LIN {X 0,Y 687.09,Z 992.261,A -85,B 0,C 180,E1 4203.082,E2 4203.082} C_VEL
LIN {X 0,Y 685.189,Z 1030.592,A -85,B 0,C 180,E1 4205.694,E2 4205.694} C_VEL
LIN {X 0,Y 683.437,Z 1066.226,A -85,B 0,C 180,E1 4208.838,E2 4208.838} C_VEL
LIN {X 0,Y 682.212,Z 1095.925,A -85,B 0,C 180,E1 4212.224,E2 4212.224} C_VEL
LIN {X 0,Y 681.417,Z 1120.366,A -85,B 0,C 180,E1 4215.88,E2 4215.88} C_VEL
LIN {X 0,Y 680.982,Z 1137.956,A -85,B 0,C 180,E1 4219.451,E2 4219.451} C_VEL
LIN {X 0,Y 680.83,Z 1150.116,A -85,B 0,C 180,E1 4222.988,E2 4222.988} C_VEL
LIN {X 0,Y 680.781,Z 1156.664,A -85,B 0,C 180,E1 4226.181,E2 4226.181} C_VEL
LIN {X 0,Y 680.724,Z 1159.5,A -85,B 0,C 180,E1 4229.999,E2 4229.999} C_VEL
LIN {X 0,Y 680.746,Z 1156.667,A -85,B 0,C 180,E1 4233.818,E2 4233.818} C_VEL
LIN {X 0,Y 680.9,Z 1150.12,A -85,B 0,C 180,E1 4237.01,E2 4237.01} C_VEL
LIN {X 0,Y 681.026,Z 1137.964,A -85,B 0,C 180,E1 4240.547,E2 4240.547} C_VEL
LIN {X 0,Y 681.455,Z 1120.372,A -85,B 0,C 180,E1 4244.117,E2 4244.117} C_VEL
LIN {X 0,Y 682.306,Z 1095.708,A -85,B 0,C 180,E1 4247.801,E2 4247.801} C_VEL
LIN {X 0,Y 683.582,Z 1064.828,A -85,B 0,C 180,E1 4251.298,E2 4251.298} C_VEL
LIN {X 0,Y 685.214,Z 1030.571,A -85,B 0,C 180,E1 4254.307,E2 4254.307} C_VEL
LIN {X 0,Y 687.123,Z 990.6,A -85,B 0,C 180,E1 4257.023,E2 4257.023} C_VEL
LIN {X 0,Y 689.048,Z 948.933,A -85,B 0,C 180,E1 4259.157,E2 4259.157} C_VEL
LIN {X 0,Y 690.718,Z 906.278,A -85,B 0,C 180,E1 4260.75,E2 4260.75} C_VEL
LIN {X 0,Y 691.991,Z 863.04,A -85,B 0,C 180,E1 4261.837,E2 4261.837} C_VEL
LIN {X 0,Y 691.945,Z 806.371,A -85,B 0,C 180,E1 4262.655,E2 4262.655} C_VEL
LIN {X 0,Y 680.359,Z 780.81,A -85,B 0,C 180,E1 4263.619,E2 4263.619} C_VEL
LIN {X 0,Y 680.153,Z 780.81,A -85,B 0,C 180,E1 4268.974,E2 4268.974} C_VEL
LIN {X 0,Y 680.422,Z 780.81,A -85,B 0,C 180,E1 4273.507,E2 4273.507} C_VEL
LIN {X 0,Y 680.172,Z 780.81,A -85,B 0,C 180,E1 4279.056,E2 4279.056} C_VEL
LIN {X 0,Y 680.227,Z 780.81,A -85,B 0,C 180,E1 4283.154,E2 4283.154} C_VEL
LIN {X 0,Y 680.191,Z 780.81,A -85,B 0,C 180,E1 4287.788,E2 4287.788} C_VEL
LIN {X 0,Y 680.45,Z 780.81,A -85,B 0,C 180,E1 4292.658,E2 4292.658} C_VEL
LIN {X 0,Y 680.425,Z 780.81,A -85,B 0,C 180,E1 4297.825,E2 4297.825} C_VEL
LIN {X 0,Y 680.516,Z 780.81,A -85,B 0,C 180,E1 4303.227,E2 4303.227} C_VEL
LIN {X 0,Y 680.543,Z 780.81,A -85,B 0,C 180,E1 4308.476,E2 4308.476} C_VEL
LIN {X 0,Y 680.684,Z 780.81,A -85,B 0,C 180,E1 4313.63,E2 4313.63} C_VEL
LIN {X 0,Y 680.631,Z 780.81,A -85,B 0,C 180,E1 4318.73,E2 4318.73} C_VEL
LIN {X 0,Y 680.66,Z 780.81,A -85,B 0,C 180,E1 4322.546,E2 4322.546} C_VEL
LIN {X 0,Y 680.609,Z 780.81,A -85,B 0,C 180,E1 4326.374,E2 4326.374} C_VEL
LIN {X 0,Y 680.539,Z 780.81,A -85,B 0,C 180,E1 4331.528,E2 4331.528} C_VEL
LIN {X 0,Y 680.552,Z 780.81,A -85,B 0,C 180,E1 4336.776,E2 4336.776} C_VEL
LIN {X 0,Y 680.385,Z 780.81,A -85,B 0,C 180,E1 4342.181,E2 4342.181} C_VEL
LIN {X 0,Y 680.369,Z 780.81,A -85,B 0,C 180,E1 4347.328,E2 4347.328} C_VEL
LIN {X 0,Y 680.311,Z 780.81,A -85,B 0,C 180,E1 4352.431,E2 4352.431} C_VEL
LIN {X 0,Y 680.211,Z 780.81,A -85,B 0,C 180,E1 4356.895,E2 4356.895} C_VEL
LIN {X 0,Y 680.321,Z 780.81,A -85,B 0,C 180,E1 4362.864,E2 4362.864} C_VEL
LIN {X 0,Y 680.144,Z 780.81,A -85,B 0,C 180,E1 4368.202,E2 4368.202} C_VEL
LIN {X 0,Y 680.322,Z 780.81,A -85,B 0,C 180,E1 4373.152,E2 4373.152} C_VEL
LIN {X 0,Y 680.408,Z 781.584,A -85,B 0,C 180,E1 4373.863,E2 4373.863} C_VEL
LIN {X 0,Y 692.3,Z 808.432,A -85,B 0,C 180,E1 4374.861,E2 4374.861} C_VEL
LIN {X 0,Y 691.206,Z 854.71,A -85,B 0,C 180,E1 4375.867,E2 4375.867} C_VEL
LIN {X 0,Y 689.535,Z 897.482,A -85,B 0,C 180,E1 4377.317,E2 4377.317} C_VEL
LIN {X 0,Y 687.817,Z 937.086,A -85,B 0,C 180,E1 4379.173,E2 4379.173} C_VEL
LIN {X 0,Y 685.919,Z 976.276,A -85,B 0,C 180,E1 4381.593,E2 4381.593} C_VEL
LIN {X 0,Y 684.097,Z 1013.54,A -85,B 0,C 180,E1 4384.581,E2 4384.581} C_VEL
LIN {X 0,Y 682.642,Z 1045.528,A -85,B 0,C 180,E1 4387.895,E2 4387.895} C_VEL
LIN {X 0,Y 681.64,Z 1071.691,A -85,B 0,C 180,E1 4391.418,E2 4391.418} C_VEL
LIN {X 0,Y 681.199,Z 1089.618,A -85,B 0,C 180,E1 4394.563,E2 4394.563} C_VEL
LIN {X 0,Y 680.932,Z 1103.952,A -85,B 0,C 180,E1 4397.975,E2 4397.975} C_VEL
LIN {X 0,Y 680.821,Z 1112.845,A -85,B 0,C 180,E1 4401.063,E2 4401.063} C_VEL
LIN {X 0,Y 680.722,Z 1118.621,A -85,B 0,C 180,E1 4404.906,E2 4404.906} C_VEL
LIN {X 0,Y 680.773,Z 1119.375,A -85,B 0,C 180,E1 4407.456,E2 4407.456} C_VEL
LIN {X 0,Y 680.825,Z 1115.946,A -85,B 0,C 180,E1 4411.273,E2 4411.273} C_VEL
LIN {X 0,Y 680.875,Z 1106.765,A -85,B 0,C 180,E1 4415.094,E2 4415.094} C_VEL
LIN {X 0,Y 681.054,Z 1093.102,A -85,B 0,C 180,E1 4418.614,E2 4418.614} C_VEL
LIN {X 0,Y 681.647,Z 1073.872,A -85,B 0,C 180,E1 4422.158,E2 4422.158} C_VEL
LIN {X 0,Y 682.563,Z 1047.417,A -85,B 0,C 180,E1 4425.79,E2 4425.79} C_VEL
LIN {X 0,Y 683.892,Z 1016.827,A -85,B 0,C 180,E1 4429.021,E2 4429.021} C_VEL
LIN {X 0,Y 685.562,Z 982.863,A -85,B 0,C 180,E1 4431.837,E2 4431.837} C_VEL
LIN {X 0,Y 687.416,Z 945.41,A -85,B 0,C 180,E1 4434.273,E2 4434.273} C_VEL
LIN {X 0,Y 689.372,Z 903.344,A -85,B 0,C 180,E1 4436.353,E2 4436.353} C_VEL
LIN {X 0,Y 691.019,Z 860.946,A -85,B 0,C 180,E1 4437.864,E2 4437.864} C_VEL
LIN {X 0,Y 692.216,Z 820.938,A -85,B 0,C 180,E1 4438.82,E2 4438.82} C_VEL
LIN {X 0,Y 691.723,Z 806.397,A -85,B 0,C 180,E1 4439.108,E2 4439.108} C_VEL
LIN {X 0,Y 680.353,Z 780.81,A -85,B 0,C 180,E1 4440.141,E2 4440.141} C_VEL
LIN {X 0,Y 680.26,Z 780.81,A -85,B 0,C 180,E1 4445.28,E2 4445.28} C_VEL
LIN {X 0,Y 680.117,Z 780.81,A -85,B 0,C 180,E1 4450.946,E2 4450.946} C_VEL
LIN {X 0,Y 680.316,Z 780.81,A -85,B 0,C 180,E1 4455.299,E2 4455.299} C_VEL
LIN {X 0,Y 680.19,Z 780.81,A -85,B 0,C 180,E1 4461.039,E2 4461.039} C_VEL
LIN {X 0,Y 680.175,Z 780.81,A -85,B 0,C 180,E1 4466.265,E2 4466.265} C_VEL
LIN {X 0,Y 680.318,Z 780.81,A -85,B 0,C 180,E1 4470.751,E2 4470.751} C_VEL
LIN {X 0,Y 680.406,Z 780.81,A -85,B 0,C 180,E1 4475.585,E2 4475.585} C_VEL
LIN {X 0,Y 680.489,Z 780.81,A -85,B 0,C 180,E1 4480.545,E2 4480.545} C_VEL
LIN {X 0,Y 680.5,Z 780.81,A -85,B 0,C 180,E1 4485.862,E2 4485.862} C_VEL
LIN {X 0,Y 680.619,Z 780.81,A -85,B 0,C 180,E1 4491.059,E2 4491.059} C_VEL
LIN {X 0,Y 680.741,Z 780.81,A -85,B 0,C 180,E1 4496.18,E2 4496.18} C_VEL
LIN {X 0,Y 680.88,Z 780.81,A -85,B 0,C 180,E1 4501.27,E2 4501.27} C_VEL
LIN {X 0,Y 680.579,Z 780.81,A -85,B 0,C 180,E1 4506.371,E2 4506.371} C_VEL
LIN {X 0,Y 680.539,Z 780.81,A -85,B 0,C 180,E1 4511.524,E2 4511.524} C_VEL
LIN {X 0,Y 680.564,Z 780.81,A -85,B 0,C 180,E1 4516.772,E2 4516.772} C_VEL
LIN {X 0,Y 680.422,Z 780.81,A -85,B 0,C 180,E1 4522.175,E2 4522.175} C_VEL
LIN {X 0,Y 680.366,Z 780.81,A -85,B 0,C 180,E1 4522.914,E2 4522.914} C_VEL
LIN {X 0,Y 676.415,Z 780.81,A -85,B 0,C 180,E1 4524.348,E2 4524.348} C_VEL
LIN {X 0,Y 672.467,Z 780.81,A -85,B 0,C 180,E1 4525.798,E2 4525.798} C_VEL
LIN {X 0,Y 672.401,Z 780.81,A -85,B 0,C 180,E1 4531.351,E2 4531.351} C_VEL
LIN {X 0,Y 672.326,Z 780.81,A -85,B 0,C 180,E1 4535.988,E2 4535.988} C_VEL
LIN {X 0,Y 672.186,Z 780.81,A -85,B 0,C 180,E1 4540.676,E2 4540.676} C_VEL
LIN {X 0,Y 672.254,Z 780.81,A -85,B 0,C 180,E1 4545.984,E2 4545.984} C_VEL
LIN {X 0,Y 672.227,Z 780.81,A -85,B 0,C 180,E1 4550.992,E2 4550.992} C_VEL
LIN {X 0,Y 672.468,Z 781.462,A -85,B 0,C 180,E1 4555.963,E2 4555.963} C_VEL
LIN {X 0,Y 685.899,Z 811.043,A -85,B 0,C 180,E1 4557.078,E2 4557.078} C_VEL
LIN {X 0,Y 685.2,Z 867.047,A -85,B 0,C 180,E1 4557.895,E2 4557.895} C_VEL
LIN {X 0,Y 683.792,Z 911.293,A -85,B 0,C 180,E1 4559.07,E2 4559.07} C_VEL
LIN {X 0,Y 681.813,Z 953.795,A -85,B 0,C 180,E1 4560.736,E2 4560.736} C_VEL
LIN {X 0,Y 679.857,Z 992.661,A -85,B 0,C 180,E1 4562.798,E2 4562.798} C_VEL
LIN {X 0,Y 677.754,Z 1031.108,A -85,B 0,C 180,E1 4565.453,E2 4565.453} C_VEL
LIN {X 0,Y 675.905,Z 1065.391,A -85,B 0,C 180,E1 4568.503,E2 4568.503} C_VEL
LIN {X 0,Y 674.501,Z 1095.923,A -85,B 0,C 180,E1 4572.014,E2 4572.014} C_VEL
LIN {X 0,Y 673.612,Z 1120.364,A -85,B 0,C 180,E1 4575.713,E2 4575.713} C_VEL
LIN {X 0,Y 673.147,Z 1136.615,A -85,B 0,C 180,E1 4578.999,E2 4578.999} C_VEL
LIN {X 0,Y 672.935,Z 1148.221,A -85,B 0,C 180,E1 4582.256,E2 4582.256} C_VEL
LIN {X 0,Y 672.913,Z 1155.686,A -85,B 0,C 180,E1 4585.491,E2 4585.491} C_VEL
LIN {X 0,Y 672.874,Z 1159.169,A -85,B 0,C 180,E1 4588.712,E2 4588.712} C_VEL
LIN {X 0,Y 672.847,Z 1158.224,A -85,B 0,C 180,E1 4592.574,E2 4592.574} C_VEL
LIN {X 0,Y 672.976,Z 1153.237,A -85,B 0,C 180,E1 4595.799,E2 4595.799} C_VEL
LIN {X 0,Y 673.038,Z 1141.814,A -85,B 0,C 180,E1 4599.693,E2 4599.693} C_VEL
LIN {X 0,Y 673.402,Z 1127.472,A -85,B 0,C 180,E1 4602.967,E2 4602.967} C_VEL
LIN {X 0,Y 674.051,Z 1105.875,A -85,B 0,C 180,E1 4606.608,E2 4606.608} C_VEL
LIN {X 0,Y 675.147,Z 1079.569,A -85,B 0,C 180,E1 4609.975,E2 4609.975} C_VEL
LIN {X 0,Y 676.765,Z 1049.45,A -85,B 0,C 180,E1 4613,E2 4613} C_VEL
LIN {X 0,Y 678.651,Z 1014.986,A -85,B 0,C 180,E1 4615.744,E2 4615.744} C_VEL
LIN {X 0,Y 680.85,Z 974.62,A -85,B 0,C 180,E1 4618.232,E2 4618.232} C_VEL
LIN {X 0,Y 682.963,Z 931.607,A -85,B 0,C 180,E1 4620.204,E2 4620.204} C_VEL
LIN {X 0,Y 684.568,Z 890.233,A -85,B 0,C 180,E1 4621.55,E2 4621.55} C_VEL
LIN {X 0,Y 685.646,Z 849.593,A -85,B 0,C 180,E1 4622.422,E2 4622.422} C_VEL
LIN {X 0,Y 685.428,Z 809.206,A -85,B 0,C 180,E1 4622.97,E2 4622.97} C_VEL
LIN {X 0,Y 672.415,Z 780.81,A -85,B 0,C 180,E1 4624.066,E2 4624.066} C_VEL
LIN {X 0,Y 672.257,Z 780.81,A -85,B 0,C 180,E1 4629.004,E2 4629.004} C_VEL
LIN {X 0,Y 672.483,Z 780.81,A -85,B 0,C 180,E1 4634.153,E2 4634.153} C_VEL
LIN {X 0,Y 672.314,Z 780.81,A -85,B 0,C 180,E1 4639.834,E2 4639.834} C_VEL
LIN {X 0,Y 672.292,Z 780.81,A -85,B 0,C 180,E1 4644.249,E2 4644.249} C_VEL
LIN {X 0,Y 672.295,Z 780.81,A -85,B 0,C 180,E1 4648.879,E2 4648.879} C_VEL
LIN {X 0,Y 672.521,Z 780.81,A -85,B 0,C 180,E1 4653.995,E2 4653.995} C_VEL
LIN {X 0,Y 672.529,Z 780.81,A -85,B 0,C 180,E1 4658.936,E2 4658.936} C_VEL
LIN {X 0,Y 672.629,Z 780.81,A -85,B 0,C 180,E1 4664.365,E2 4664.365} C_VEL
LIN {X 0,Y 672.708,Z 780.81,A -85,B 0,C 180,E1 4669.651,E2 4669.651} C_VEL
LIN {X 0,Y 672.703,Z 780.81,A -85,B 0,C 180,E1 4674.848,E2 4674.848} C_VEL
LIN {X 0,Y 672.744,Z 780.81,A -85,B 0,C 180,E1 4678.715,E2 4678.715} C_VEL
LIN {X 0,Y 672.758,Z 780.81,A -85,B 0,C 180,E1 4682.576,E2 4682.576} C_VEL
LIN {X 0,Y 672.702,Z 780.81,A -85,B 0,C 180,E1 4686.45,E2 4686.45} C_VEL
LIN {X 0,Y 672.681,Z 780.81,A -85,B 0,C 180,E1 4690.353,E2 4690.353} C_VEL
LIN {X 0,Y 672.653,Z 780.81,A -85,B 0,C 180,E1 4695.638,E2 4695.638} C_VEL
LIN {X 0,Y 672.522,Z 780.81,A -85,B 0,C 180,E1 4701.068,E2 4701.068} C_VEL
LIN {X 0,Y 672.434,Z 780.81,A -85,B 0,C 180,E1 4706.705,E2 4706.705} C_VEL
LIN {X 0,Y 672.359,Z 780.81,A -85,B 0,C 180,E1 4711.348,E2 4711.348} C_VEL
LIN {X 0,Y 672.303,Z 780.81,A -85,B 0,C 180,E1 4715.988,E2 4715.988} C_VEL
LIN {X 0,Y 672.208,Z 780.81,A -85,B 0,C 180,E1 4720.68,E2 4720.68} C_VEL
LIN {X 0,Y 672.349,Z 780.81,A -85,B 0,C 180,E1 4725.981,E2 4725.981} C_VEL
LIN {X 0,Y 672.42,Z 780.81,A -85,B 0,C 180,E1 4731.854,E2 4731.854} C_VEL
LIN {X 0,Y 672.432,Z 780.81,A -85,B 0,C 180,E1 4733.398,E2 4733.398} C_VEL
LIN {X 0,Y 685.61,Z 812.911,A -85,B 0,C 180,E1 4734.594,E2 4734.594} C_VEL
LIN {X 0,Y 684.35,Z 856.364,A -85,B 0,C 180,E1 4735.567,E2 4735.567} C_VEL
LIN {X 0,Y 682.476,Z 899.679,A -85,B 0,C 180,E1 4737.073,E2 4737.073} C_VEL
LIN {X 0,Y 680.432,Z 940.833,A -85,B 0,C 180,E1 4739.065,E2 4739.065} C_VEL
LIN {X 0,Y 678.453,Z 978.628,A -85,B 0,C 180,E1 4741.469,E2 4741.469} C_VEL
LIN {X 0,Y 676.521,Z 1014.57,A -85,B 0,C 180,E1 4744.413,E2 4744.413} C_VEL
LIN {X 0,Y 674.916,Z 1046.522,A -85,B 0,C 180,E1 4747.785,E2 4747.785} C_VEL
LIN {X 0,Y 673.823,Z 1072.54,A -85,B 0,C 180,E1 4751.364,E2 4751.364} C_VEL
LIN {X 0,Y 673.302,Z 1091.329,A -85,B 0,C 180,E1 4754.78,E2 4754.78} C_VEL
LIN {X 0,Y 673.042,Z 1105.621,A -85,B 0,C 180,E1 4758.343,E2 4758.343} C_VEL
LIN {X 0,Y 672.916,Z 1115.336,A -85,B 0,C 180,E1 4762.257,E2 4762.257} C_VEL
LIN {X 0,Y 672.898,Z 1119.294,A -85,B 0,C 180,E1 4766.138,E2 4766.138} C_VEL
LIN {X 0,Y 672.908,Z 1117.744,A -85,B 0,C 180,E1 4770.001,E2 4770.001} C_VEL
LIN {X 0,Y 673.061,Z 1110.564,A -85,B 0,C 180,E1 4773.863,E2 4773.863} C_VEL
LIN {X 0,Y 673.213,Z 1097.492,A -85,B 0,C 180,E1 4777.741,E2 4777.741} C_VEL
LIN {X 0,Y 673.691,Z 1079.897,A -85,B 0,C 180,E1 4781.319,E2 4781.319} C_VEL
LIN {X 0,Y 674.447,Z 1056.011,A -85,B 0,C 180,E1 4784.932,E2 4784.932} C_VEL
LIN {X 0,Y 675.9,Z 1025.8,A -85,B 0,C 180,E1 4788.409,E2 4788.409} C_VEL
LIN {X 0,Y 677.806,Z 990.093,A -85,B 0,C 180,E1 4791.584,E2 4791.584} C_VEL
LIN {X 0,Y 679.981,Z 950.7,A -85,B 0,C 180,E1 4794.278,E2 4794.278} C_VEL
LIN {X 0,Y 682.058,Z 909.948,A -85,B 0,C 180,E1 4796.391,E2 4796.391} C_VEL
LIN {X 0,Y 683.81,Z 870.24,A -85,B 0,C 180,E1 4797.919,E2 4797.919} C_VEL
LIN {X 0,Y 685.308,Z 826.609,A -85,B 0,C 180,E1 4799.065,E2 4799.065} C_VEL
LIN {X 0,Y 684.896,Z 808.687,A -85,B 0,C 180,E1 4799.434,E2 4799.434} C_VEL
LIN {X 0,Y 672.411,Z 780.81,A -85,B 0,C 180,E1 4800.538,E2 4800.538} C_VEL
LIN {X 0,Y 672.289,Z 780.81,A -85,B 0,C 180,E1 4805.762,E2 4805.762} C_VEL
LIN {X 0,Y 672.207,Z 780.81,A -85,B 0,C 180,E1 4810.687,E2 4810.687} C_VEL
LIN {X 0,Y 672.336,Z 780.81,A -85,B 0,C 180,E1 4815.841,E2 4815.841} C_VEL
LIN {X 0,Y 672.293,Z 780.81,A -85,B 0,C 180,E1 4821.003,E2 4821.003} C_VEL
LIN {X 0,Y 672.283,Z 780.81,A -85,B 0,C 180,E1 4826.271,E2 4826.271} C_VEL
LIN {X 0,Y 672.462,Z 780.81,A -85,B 0,C 180,E1 4831.846,E2 4831.846} C_VEL
LIN {X 0,Y 672.461,Z 780.81,A -85,B 0,C 180,E1 4837.122,E2 4837.122} C_VEL
LIN {X 0,Y 672.59,Z 780.81,A -85,B 0,C 180,E1 4841.668,E2 4841.668} C_VEL
LIN {X 0,Y 672.588,Z 780.81,A -85,B 0,C 180,E1 4845.692,E2 4845.692} C_VEL
LIN {X 0,Y 672.713,Z 780.81,A -85,B 0,C 180,E1 4851.256,E2 4851.256} C_VEL
LIN {X 0,Y 672.831,Z 780.81,A -85,B 0,C 180,E1 4856.135,E2 4856.135} C_VEL
LIN {X 0,Y 672.979,Z 780.81,A -85,B 0,C 180,E1 4861.284,E2 4861.284} C_VEL
LIN {X 0,Y 672.674,Z 780.81,A -85,B 0,C 180,E1 4866.446,E2 4866.446} C_VEL
LIN {X 0,Y 672.669,Z 780.81,A -85,B 0,C 180,E1 4870.349,E2 4870.349} C_VEL
LIN {X 0,Y 672.647,Z 780.81,A -85,B 0,C 180,E1 4875.635,E2 4875.635} C_VEL
LIN {X 0,Y 672.572,Z 780.81,A -85,B 0,C 180,E1 4881.062,E2 4881.062} C_VEL
LIN {X 0,Y 672.467,Z 780.81,A -85,B 0,C 180,E1 4885.798,E2 4885.798} C_VEL
LIN {X 0,Y 668.561,Z 780.81,A -85,B 0,C 180,E1 4887.256,E2 4887.256} C_VEL
LIN {X 0,Y 664.506,Z 780.81,A -85,B 0,C 180,E1 4888.73,E2 4888.73} C_VEL
LIN {X 0,Y 664.534,Z 780.81,A -85,B 0,C 180,E1 4893.067,E2 4893.067} C_VEL
LIN {X 0,Y 664.329,Z 780.81,A -85,B 0,C 180,E1 4897.88,E2 4897.88} C_VEL
LIN {X 0,Y 664.274,Z 780.81,A -85,B 0,C 180,E1 4903.285,E2 4903.285} C_VEL
LIN {X 0,Y 664.27,Z 780.81,A -85,B 0,C 180,E1 4908.722,E2 4908.722} C_VEL
LIN {X 0,Y 664.417,Z 780.81,A -85,B 0,C 180,E1 4913.748,E2 4913.748} C_VEL
LIN {X 0,Y 664.48,Z 780.81,A -85,B 0,C 180,E1 4915.49,E2 4915.49} C_VEL
LIN {X 0,Y 679.318,Z 813.462,A -85,B 0,C 180,E1 4916.747,E2 4916.747} C_VEL
LIN {X 0,Y 678.502,Z 867.045,A -85,B 0,C 180,E1 4917.539,E2 4917.539} C_VEL
LIN {X 0,Y 676.925,Z 911.802,A -85,B 0,C 180,E1 4918.739,E2 4918.739} C_VEL
LIN {X 0,Y 674.776,Z 954.064,A -85,B 0,C 180,E1 4920.414,E2 4920.414} C_VEL
LIN {X 0,Y 672.573,Z 994.032,A -85,B 0,C 180,E1 4922.568,E2 4922.568} C_VEL
LIN {X 0,Y 670.323,Z 1031.236,A -85,B 0,C 180,E1 4925.173,E2 4925.173} C_VEL
LIN {X 0,Y 668.273,Z 1066.264,A -85,B 0,C 180,E1 4928.338,E2 4928.338} C_VEL
LIN {X 0,Y 666.779,Z 1096.55,A -85,B 0,C 180,E1 4931.882,E2 4931.882} C_VEL
LIN {X 0,Y 665.808,Z 1120.363,A -85,B 0,C 180,E1 4935.542,E2 4935.542} C_VEL
LIN {X 0,Y 665.248,Z 1137.958,A -85,B 0,C 180,E1 4939.198,E2 4939.198} C_VEL
LIN {X 0,Y 665.055,Z 1150.116,A -85,B 0,C 180,E1 4942.82,E2 4942.82} C_VEL
LIN {X 0,Y 664.989,Z 1156.663,A -85,B 0,C 180,E1 4946.09,E2 4946.09} C_VEL
LIN {X 0,Y 664.947,Z 1159.5,A -85,B 0,C 180,E1 4949.999,E2 4949.999} C_VEL
LIN {X 0,Y 664.964,Z 1156.666,A -85,B 0,C 180,E1 4953.908,E2 4953.908} C_VEL
LIN {X 0,Y 665.132,Z 1150.12,A -85,B 0,C 180,E1 4957.177,E2 4957.177} C_VEL
LIN {X 0,Y 665.406,Z 1136.623,A -85,B 0,C 180,E1 4961.129,E2 4961.129} C_VEL
LIN {X 0,Y 665.961,Z 1118.841,A -85,B 0,C 180,E1 4964.717,E2 4964.717} C_VEL
LIN {X 0,Y 666.903,Z 1095.045,A -85,B 0,C 180,E1 4968.311,E2 4968.311} C_VEL
LIN {X 0,Y 668.399,Z 1064.744,A -85,B 0,C 180,E1 4971.815,E2 4971.815} C_VEL
LIN {X 0,Y 670.485,Z 1029.076,A -85,B 0,C 180,E1 4974.997,E2 4974.997} C_VEL
LIN {X 0,Y 672.77,Z 990.127,A -85,B 0,C 180,E1 4977.678,E2 4977.678} C_VEL
LIN {X 0,Y 675.203,Z 947.105,A -85,B 0,C 180,E1 4979.903,E2 4979.903} C_VEL
LIN {X 0,Y 677.144,Z 904.152,A -85,B 0,C 180,E1 4981.507,E2 4981.507} C_VEL
LIN {X 0,Y 678.642,Z 860.929,A -85,B 0,C 180,E1 4982.58,E2 4982.58} C_VEL
LIN {X 0,Y 678.651,Z 811.393,A -85,B 0,C 180,E1 4983.315,E2 4983.315} C_VEL
LIN {X 0,Y 664.443,Z 780.81,A -85,B 0,C 180,E1 4984.511,E2 4984.511} C_VEL
LIN {X 0,Y 664.333,Z 780.81,A -85,B 0,C 180,E1 4989.56,E2 4989.56} C_VEL
LIN {X 0,Y 664.474,Z 780.81,A -85,B 0,C 180,E1 4994.827,E2 4994.827} C_VEL
LIN {X 0,Y 664.395,Z 780.81,A -85,B 0,C 180,E1 5000.65,E2 5000.65} C_VEL
LIN {X 0,Y 664.346,Z 780.81,A -85,B 0,C 180,E1 5005.354,E2 5005.354} C_VEL
LIN {X 0,Y 664.408,Z 780.81,A -85,B 0,C 180,E1 5009.984,E2 5009.984} C_VEL
LIN {X 0,Y 664.606,Z 780.81,A -85,B 0,C 180,E1 5014.412,E2 5014.412} C_VEL
LIN {X 0,Y 664.627,Z 780.81,A -85,B 0,C 180,E1 5020.065,E2 5020.065} C_VEL
LIN {X 0,Y 664.658,Z 780.81,A -85,B 0,C 180,E1 5025.522,E2 5025.522} C_VEL
LIN {X 0,Y 664.759,Z 780.81,A -85,B 0,C 180,E1 5030.848,E2 5030.848} C_VEL
LIN {X 0,Y 664.919,Z 780.81,A -85,B 0,C 180,E1 5036.093,E2 5036.093} C_VEL
LIN {X 0,Y 665.057,Z 780.81,A -85,B 0,C 180,E1 5041.333,E2 5041.333} C_VEL
LIN {X 0,Y 664.802,Z 780.81,A -85,B 0,C 180,E1 5046.527,E2 5046.527} C_VEL
LIN {X 0,Y 664.723,Z 780.81,A -85,B 0,C 180,E1 5051.806,E2 5051.806} C_VEL
LIN {X 0,Y 664.702,Z 780.81,A -85,B 0,C 180,E1 5057.293,E2 5057.293} C_VEL
LIN {X 0,Y 664.539,Z 780.81,A -85,B 0,C 180,E1 5062.739,E2 5062.739} C_VEL
LIN {X 0,Y 664.503,Z 780.81,A -85,B 0,C 180,E1 5067.519,E2 5067.519} C_VEL
LIN {X 0,Y 664.506,Z 780.81,A -85,B 0,C 180,E1 5073.073,E2 5073.073} C_VEL
LIN {X 0,Y 664.317,Z 780.81,A -85,B 0,C 180,E1 5077.886,E2 5077.886} C_VEL
LIN {X 0,Y 664.433,Z 780.81,A -85,B 0,C 180,E1 5083.301,E2 5083.301} C_VEL
LIN {X 0,Y 664.315,Z 780.81,A -85,B 0,C 180,E1 5088.727,E2 5088.727} C_VEL
LIN {X 0,Y 664.51,Z 780.81,A -85,B 0,C 180,E1 5092.933,E2 5092.933} C_VEL
LIN {X 0,Y 678.862,Z 813.526,A -85,B 0,C 180,E1 5094.244,E2 5094.244} C_VEL
LIN {X 0,Y 677.544,Z 857.036,A -85,B 0,C 180,E1 5095.234,E2 5095.234} C_VEL
LIN {X 0,Y 675.456,Z 901.471,A -85,B 0,C 180,E1 5096.808,E2 5096.808} C_VEL
LIN {X 0,Y 673.206,Z 942.54,A -85,B 0,C 180,E1 5098.841,E2 5098.841} C_VEL
LIN {X 0,Y 671.047,Z 979.928,A -85,B 0,C 180,E1 5101.269,E2 5101.269} C_VEL
LIN {X 0,Y 668.947,Z 1015.39,A -85,B 0,C 180,E1 5104.225,E2 5104.225} C_VEL
LIN {X 0,Y 667.242,Z 1046.933,A -85,B 0,C 180,E1 5107.608,E2 5107.608} C_VEL
LIN {X 0,Y 666.017,Z 1073.389,A -85,B 0,C 180,E1 5111.309,E2 5111.309} C_VEL
LIN {X 0,Y 665.453,Z 1091.617,A -85,B 0,C 180,E1 5114.696,E2 5114.696} C_VEL
LIN {X 0,Y 665.154,Z 1105.491,A -85,B 0,C 180,E1 5118.203,E2 5118.203} C_VEL
LIN {X 0,Y 665.031,Z 1114.316,A -85,B 0,C 180,E1 5121.647,E2 5121.647} C_VEL
LIN {X 0,Y 664.942,Z 1118.565,A -85,B 0,C 180,E1 5124.785,E2 5124.785} C_VEL
LIN {X 0,Y 664.928,Z 1118.896,A -85,B 0,C 180,E1 5128.699,E2 5128.699} C_VEL
LIN {X 0,Y 665.042,Z 1113.683,A -85,B 0,C 180,E1 5132.605,E2 5132.605} C_VEL
LIN {X 0,Y 665.178,Z 1103.789,A -85,B 0,C 180,E1 5136.195,E2 5136.195} C_VEL
LIN {X 0,Y 665.545,Z 1088.871,A -85,B 0,C 180,E1 5139.805,E2 5139.805} C_VEL
LIN {X 0,Y 666.435,Z 1066.853,A -85,B 0,C 180,E1 5143.607,E2 5143.607} C_VEL
LIN {X 0,Y 667.627,Z 1040.003,A -85,B 0,C 180,E1 5147.113,E2 5147.113} C_VEL
LIN {X 0,Y 669.189,Z 1010.456,A -85,B 0,C 180,E1 5150.139,E2 5150.139} C_VEL
LIN {X 0,Y 671.381,Z 974.686,A -85,B 0,C 180,E1 5153.021,E2 5153.021} C_VEL
LIN {X 0,Y 673.765,Z 934.374,A -85,B 0,C 180,E1 5155.525,E2 5155.525} C_VEL
LIN {X 0,Y 675.975,Z 889.563,A -85,B 0,C 180,E1 5157.592,E2 5157.592} C_VEL
LIN {X 0,Y 678.044,Z 842.209,A -85,B 0,C 180,E1 5159.074,E2 5159.074} C_VEL
LIN {X 0,Y 678.295,Z 811.523,A -85,B 0,C 180,E1 5159.735,E2 5159.735} C_VEL
LIN {X 0,Y 664.478,Z 780.81,A -85,B 0,C 180,E1 5161.035,E2 5161.035} C_VEL
LIN {X 0,Y 664.38,Z 780.81,A -85,B 0,C 180,E1 5166.254,E2 5166.254} C_VEL
LIN {X 0,Y 664.323,Z 780.81,A -85,B 0,C 180,E1 5171.363,E2 5171.363} C_VEL
LIN {X 0,Y 664.316,Z 780.81,A -85,B 0,C 180,E1 5176.711,E2 5176.711} C_VEL
LIN {X 0,Y 664.334,Z 780.81,A -85,B 0,C 180,E1 5182.115,E2 5182.115} C_VEL
LIN {X 0,Y 664.373,Z 780.81,A -85,B 0,C 180,E1 5187.306,E2 5187.306} C_VEL
LIN {X 0,Y 664.584,Z 780.81,A -85,B 0,C 180,E1 5192.954,E2 5192.954} C_VEL
LIN {X 0,Y 664.607,Z 780.81,A -85,B 0,C 180,E1 5198.669,E2 5198.669} C_VEL
LIN {X 0,Y 664.733,Z 780.81,A -85,B 0,C 180,E1 5204.17,E2 5204.17} C_VEL
LIN {X 0,Y 664.821,Z 780.81,A -85,B 0,C 180,E1 5209.523,E2 5209.523} C_VEL
LIN {X 0,Y 664.823,Z 780.81,A -85,B 0,C 180,E1 5214.782,E2 5214.782} C_VEL
LIN {X 0,Y 664.903,Z 780.81,A -85,B 0,C 180,E1 5219.705,E2 5219.705} C_VEL
LIN {X 0,Y 664.928,Z 780.81,A -85,B 0,C 180,E1 5223.907,E2 5223.907} C_VEL
LIN {X 0,Y 664.856,Z 780.81,A -85,B 0,C 180,E1 5229.151,E2 5229.151} C_VEL
LIN {X 0,Y 664.693,Z 780.81,A -85,B 0,C 180,E1 5234.477,E2 5234.477} C_VEL
LIN {X 0,Y 664.701,Z 780.81,A -85,B 0,C 180,E1 5238.553,E2 5238.553} C_VEL
LIN {X 0,Y 664.578,Z 780.81,A -85,B 0,C 180,E1 5242.733,E2 5242.733} C_VEL
LIN {X 0,Y 664.539,Z 780.81,A -85,B 0,C 180,E1 5247.521,E2 5247.521} C_VEL
LIN {X 0,Y 664.506,Z 780.81,A -85,B 0,C 180,E1 5248.73,E2 5248.73} C_VEL
LIN {X 0,Y 660.531,Z 780.81,A -85,B 0,C 180,E1 5250.205,E2 5250.205} C_VEL
LIN {X 0,Y 656.622,Z 780.81,A -85,B 0,C 180,E1 5251.697,E2 5251.697} C_VEL
LIN {X 0,Y 656.493,Z 780.81,A -85,B 0,C 180,E1 5256.75,E2 5256.75} C_VEL
LIN {X 0,Y 656.328,Z 780.81,A -85,B 0,C 180,E1 5262.543,E2 5262.543} C_VEL
LIN {X 0,Y 656.328,Z 780.81,A -85,B 0,C 180,E1 5268.11,E2 5268.11} C_VEL
LIN {X 0,Y 656.53,Z 780.81,A -85,B 0,C 180,E1 5273.649,E2 5273.649} C_VEL
LIN {X 0,Y 656.569,Z 780.81,A -85,B 0,C 180,E1 5275.002,E2 5275.002} C_VEL
LIN {X 0,Y 672.73,Z 816.005,A -85,B 0,C 180,E1 5276.411,E2 5276.411} C_VEL
LIN {X 0,Y 671.792,Z 868.139,A -85,B 0,C 180,E1 5277.201,E2 5277.201} C_VEL
LIN {X 0,Y 670.071,Z 912.744,A -85,B 0,C 180,E1 5278.414,E2 5278.414} C_VEL
LIN {X 0,Y 667.668,Z 956.622,A -85,B 0,C 180,E1 5280.193,E2 5280.193} C_VEL
LIN {X 0,Y 665.273,Z 996.002,A -85,B 0,C 180,E1 5282.372,E2 5282.372} C_VEL
LIN {X 0,Y 662.87,Z 1032.282,A -85,B 0,C 180,E1 5284.965,E2 5284.965} C_VEL
LIN {X 0,Y 660.654,Z 1066.853,A -85,B 0,C 180,E1 5288.14,E2 5288.14} C_VEL
LIN {X 0,Y 659.137,Z 1096.123,A -85,B 0,C 180,E1 5291.606,E2 5291.606} C_VEL
LIN {X 0,Y 658.032,Z 1120.362,A -85,B 0,C 180,E1 5295.368,E2 5295.368} C_VEL
LIN {X 0,Y 657.385,Z 1137.957,A -85,B 0,C 180,E1 5299.067,E2 5299.067} C_VEL
LIN {X 0,Y 657.165,Z 1150.116,A -85,B 0,C 180,E1 5302.734,E2 5302.734} C_VEL
LIN {X 0,Y 657.09,Z 1156.663,A -85,B 0,C 180,E1 5306.043,E2 5306.043} C_VEL
LIN {X 0,Y 657.07,Z 1159.5,A -85,B 0,C 180,E1 5309.999,E2 5309.999} C_VEL
LIN {X 0,Y 657.066,Z 1156.665,A -85,B 0,C 180,E1 5313.955,E2 5313.955} C_VEL
LIN {X 0,Y 657.244,Z 1150.12,A -85,B 0,C 180,E1 5317.264,E2 5317.264} C_VEL
LIN {X 0,Y 657.469,Z 1137.964,A -85,B 0,C 180,E1 5320.93,E2 5320.93} C_VEL
LIN {X 0,Y 658.073,Z 1120.368,A -85,B 0,C 180,E1 5324.63,E2 5324.63} C_VEL
LIN {X 0,Y 659.127,Z 1096.443,A -85,B 0,C 180,E1 5328.351,E2 5328.351} C_VEL
LIN {X 0,Y 660.739,Z 1066.895,A -85,B 0,C 180,E1 5331.853,E2 5331.853} C_VEL
LIN {X 0,Y 662.925,Z 1032.303,A -85,B 0,C 180,E1 5335.031,E2 5335.031} C_VEL
LIN {X 0,Y 665.242,Z 995.514,A -85,B 0,C 180,E1 5337.662,E2 5337.662} C_VEL
LIN {X 0,Y 667.696,Z 956.653,A -85,B 0,C 180,E1 5339.803,E2 5339.803} C_VEL
LIN {X 0,Y 669.999,Z 912.617,A -85,B 0,C 180,E1 5341.594,E2 5341.594} C_VEL
LIN {X 0,Y 671.823,Z 866.449,A -85,B 0,C 180,E1 5342.838,E2 5342.838} C_VEL
LIN {X 0,Y 672.072,Z 814.09,A -85,B 0,C 180,E1 5343.649,E2 5343.649} C_VEL
LIN {X 0,Y 656.503,Z 780.81,A -85,B 0,C 180,E1 5345.042,E2 5345.042} C_VEL
LIN {X 0,Y 656.401,Z 780.81,A -85,B 0,C 180,E1 5350.577,E2 5350.577} C_VEL
LIN {X 0,Y 656.491,Z 780.81,A -85,B 0,C 180,E1 5355.524,E2 5355.524} C_VEL
LIN {X 0,Y 656.429,Z 780.81,A -85,B 0,C 180,E1 5361.506,E2 5361.506} C_VEL
LIN {X 0,Y 656.397,Z 780.81,A -85,B 0,C 180,E1 5366.47,E2 5366.47} C_VEL
LIN {X 0,Y 656.566,Z 780.81,A -85,B 0,C 180,E1 5371.105,E2 5371.105} C_VEL
LIN {X 0,Y 656.656,Z 780.81,A -85,B 0,C 180,E1 5375.537,E2 5375.537} C_VEL
LIN {X 0,Y 656.731,Z 780.81,A -85,B 0,C 180,E1 5381.214,E2 5381.214} C_VEL
LIN {X 0,Y 656.744,Z 780.81,A -85,B 0,C 180,E1 5385.344,E2 5385.344} C_VEL
LIN {X 0,Y 656.859,Z 780.81,A -85,B 0,C 180,E1 5390.737,E2 5390.737} C_VEL
LIN {X 0,Y 657.008,Z 780.81,A -85,B 0,C 180,E1 5396.046,E2 5396.046} C_VEL
LIN {X 0,Y 657.188,Z 780.81,A -85,B 0,C 180,E1 5401.319,E2 5401.319} C_VEL
LIN {X 0,Y 656.895,Z 780.81,A -85,B 0,C 180,E1 5406.606,E2 5406.606} C_VEL
LIN {X 0,Y 656.843,Z 780.81,A -85,B 0,C 180,E1 5410.606,E2 5410.606} C_VEL
LIN {X 0,Y 656.816,Z 780.81,A -85,B 0,C 180,E1 5416.026,E2 5416.026} C_VEL
LIN {X 0,Y 656.653,Z 780.81,A -85,B 0,C 180,E1 5421.603,E2 5421.603} C_VEL
LIN {X 0,Y 656.564,Z 780.81,A -85,B 0,C 180,E1 5426.158,E2 5426.158} C_VEL
LIN {X 0,Y 656.574,Z 780.81,A -85,B 0,C 180,E1 5431.62,E2 5431.62} C_VEL
LIN {X 0,Y 656.445,Z 780.81,A -85,B 0,C 180,E1 5436.758,E2 5436.758} C_VEL
LIN {X 0,Y 656.455,Z 780.81,A -85,B 0,C 180,E1 5442.557,E2 5442.557} C_VEL
LIN {X 0,Y 656.374,Z 780.81,A -85,B 0,C 180,E1 5447.444,E2 5447.444} C_VEL
LIN {X 0,Y 656.61,Z 780.81,A -85,B 0,C 180,E1 5452.451,E2 5452.451} C_VEL
LIN {X 0,Y 672.175,Z 817.721,A -85,B 0,C 180,E1 5453.956,E2 5453.956} C_VEL
LIN {X 0,Y 670.727,Z 858.839,A -85,B 0,C 180,E1 5454.932,E2 5454.932} C_VEL
LIN {X 0,Y 668.441,Z 903.732,A -85,B 0,C 180,E1 5456.558,E2 5456.558} C_VEL
LIN {X 0,Y 665.925,Z 946.007,A -85,B 0,C 180,E1 5458.714,E2 5458.714} C_VEL
LIN {X 0,Y 663.44,Z 983.835,A -85,B 0,C 180,E1 5461.261,E2 5461.261} C_VEL
LIN {X 0,Y 661.348,Z 1016.769,A -85,B 0,C 180,E1 5464.089,E2 5464.089} C_VEL
LIN {X 0,Y 659.645,Z 1046.412,A -85,B 0,C 180,E1 5467.31,E2 5467.31} C_VEL
LIN {X 0,Y 658.356,Z 1072.472,A -85,B 0,C 180,E1 5470.978,E2 5470.978} C_VEL
LIN {X 0,Y 657.593,Z 1091.186,A -85,B 0,C 180,E1 5474.453,E2 5474.453} C_VEL
LIN {X 0,Y 657.291,Z 1105.361,A -85,B 0,C 180,E1 5478.06,E2 5478.06} C_VEL
LIN {X 0,Y 657.138,Z 1113.914,A -85,B 0,C 180,E1 5481.363,E2 5481.363} C_VEL
LIN {X 0,Y 657.038,Z 1118.536,A -85,B 0,C 180,E1 5484.722,E2 5484.722} C_VEL
LIN {X 0,Y 657.028,Z 1118.924,A -85,B 0,C 180,E1 5488.683,E2 5488.683} C_VEL
LIN {X 0,Y 657.144,Z 1113.75,A -85,B 0,C 180,E1 5492.637,E2 5492.637} C_VEL
LIN {X 0,Y 657.321,Z 1103.916,A -85,B 0,C 180,E1 5496.27,E2 5496.27} C_VEL
LIN {X 0,Y 657.706,Z 1089.046,A -85,B 0,C 180,E1 5499.923,E2 5499.923} C_VEL
LIN {X 0,Y 658.637,Z 1067.101,A -85,B 0,C 180,E1 5503.771,E2 5503.771} C_VEL
LIN {X 0,Y 659.964,Z 1040.332,A -85,B 0,C 180,E1 5507.318,E2 5507.318} C_VEL
LIN {X 0,Y 661.758,Z 1010.026,A -85,B 0,C 180,E1 5510.455,E2 5510.455} C_VEL
LIN {X 0,Y 664.081,Z 975.237,A -85,B 0,C 180,E1 5513.29,E2 5513.29} C_VEL
LIN {X 0,Y 666.644,Z 934.942,A -85,B 0,C 180,E1 5515.827,E2 5515.827} C_VEL
LIN {X 0,Y 669.031,Z 890.517,A -85,B 0,C 180,E1 5517.903,E2 5517.903} C_VEL
LIN {X 0,Y 671.186,Z 844.768,A -85,B 0,C 180,E1 5519.368,E2 5519.368} C_VEL
LIN {X 0,Y 671.654,Z 814.315,A -85,B 0,C 180,E1 5520.053,E2 5520.053} C_VEL
LIN {X 0,Y 656.575,Z 780.81,A -85,B 0,C 180,E1 5521.515,E2 5521.515} C_VEL
LIN {X 0,Y 656.434,Z 780.81,A -85,B 0,C 180,E1 5526.765,E2 5526.765} C_VEL
LIN {X 0,Y 656.459,Z 780.81,A -85,B 0,C 180,E1 5532.564,E2 5532.564} C_VEL
LIN {X 0,Y 656.357,Z 780.81,A -85,B 0,C 180,E1 5537.454,E2 5537.454} C_VEL
LIN {X 0,Y 656.421,Z 780.81,A -85,B 0,C 180,E1 5543.24,E2 5543.24} C_VEL
LIN {X 0,Y 656.482,Z 780.81,A -85,B 0,C 180,E1 5548.396,E2 5548.396} C_VEL
LIN {X 0,Y 656.676,Z 780.81,A -85,B 0,C 180,E1 5554.076,E2 5554.076} C_VEL
LIN {X 0,Y 656.719,Z 780.81,A -85,B 0,C 180,E1 5559.811,E2 5559.811} C_VEL
LIN {X 0,Y 656.768,Z 780.81,A -85,B 0,C 180,E1 5565.096,E2 5565.096} C_VEL
LIN {X 0,Y 656.897,Z 780.81,A -85,B 0,C 180,E1 5570.733,E2 5570.733} C_VEL
LIN {X 0,Y 657.029,Z 780.81,A -85,B 0,C 180,E1 5576.042,E2 5576.042} C_VEL
LIN {X 0,Y 657.216,Z 780.81,A -85,B 0,C 180,E1 5581.315,E2 5581.315} C_VEL
LIN {X 0,Y 656.871,Z 780.81,A -85,B 0,C 180,E1 5586.602,E2 5586.602} C_VEL
LIN {X 0,Y 656.834,Z 780.81,A -85,B 0,C 180,E1 5590.602,E2 5590.602} C_VEL
LIN {X 0,Y 656.815,Z 780.81,A -85,B 0,C 180,E1 5596.021,E2 5596.021} C_VEL
LIN {X 0,Y 656.7,Z 780.81,A -85,B 0,C 180,E1 5601.597,E2 5601.597} C_VEL
LIN {X 0,Y 656.618,Z 780.81,A -85,B 0,C 180,E1 5606.164,E2 5606.164} C_VEL
LIN {X 0,Y 656.622,Z 780.81,A -85,B 0,C 180,E1 5611.697,E2 5611.697} C_VEL
LIN {X 0,Y 652.591,Z 780.81,A -85,B 0,C 180,E1 5613.187,E2 5613.187} C_VEL
LIN {X 0,Y 648.592,Z 780.81,A -85,B 0,C 180,E1 5614.695,E2 5614.695} C_VEL
LIN {X 0,Y 648.395,Z 780.81,A -85,B 0,C 180,E1 5619.728,E2 5619.728} C_VEL
LIN {X 0,Y 648.454,Z 780.81,A -85,B 0,C 180,E1 5624.342,E2 5624.342} C_VEL
LIN {X 0,Y 648.418,Z 780.81,A -85,B 0,C 180,E1 5629.267,E2 5629.267} C_VEL
LIN {X 0,Y 648.608,Z 780.81,A -85,B 0,C 180,E1 5634.516,E2 5634.516} C_VEL
LIN {X 0,Y 666.134,Z 818.283,A -85,B 0,C 180,E1 5636.067,E2 5636.067} C_VEL
LIN {X 0,Y 665.099,Z 867.951,A -85,B 0,C 180,E1 5636.829,E2 5636.829} C_VEL
LIN {X 0,Y 663.302,Z 912.272,A -85,B 0,C 180,E1 5638.038,E2 5638.038} C_VEL
LIN {X 0,Y 660.754,Z 955.47,A -85,B 0,C 180,E1 5639.792,E2 5639.792} C_VEL
LIN {X 0,Y 658.153,Z 995.259,A -85,B 0,C 180,E1 5641.998,E2 5641.998} C_VEL
LIN {X 0,Y 655.542,Z 1032.281,A -85,B 0,C 180,E1 5644.666,E2 5644.666} C_VEL
LIN {X 0,Y 653.173,Z 1066.18,A -85,B 0,C 180,E1 5647.801,E2 5647.801} C_VEL
LIN {X 0,Y 651.397,Z 1096.819,A -85,B 0,C 180,E1 5651.477,E2 5651.477} C_VEL
LIN {X 0,Y 650.251,Z 1120.36,A -85,B 0,C 180,E1 5655.188,E2 5655.188} C_VEL
LIN {X 0,Y 649.515,Z 1137.957,A -85,B 0,C 180,E1 5658.933,E2 5658.933} C_VEL
LIN {X 0,Y 649.298,Z 1150.116,A -85,B 0,C 180,E1 5662.645,E2 5662.645} C_VEL
LIN {X 0,Y 649.193,Z 1156.662,A -85,B 0,C 180,E1 5665.995,E2 5665.995} C_VEL
LIN {X 0,Y 649.19,Z 1159.5,A -85,B 0,C 180,E1 5669.999,E2 5669.999} C_VEL
LIN {X 0,Y 649.171,Z 1156.665,A -85,B 0,C 180,E1 5674.004,E2 5674.004} C_VEL
LIN {X 0,Y 649.375,Z 1150.119,A -85,B 0,C 180,E1 5677.352,E2 5677.352} C_VEL
LIN {X 0,Y 649.675,Z 1136.625,A -85,B 0,C 180,E1 5681.402,E2 5681.402} C_VEL
LIN {X 0,Y 650.392,Z 1118.046,A -85,B 0,C 180,E1 5685.218,E2 5685.218} C_VEL
LIN {X 0,Y 651.549,Z 1094.776,A -85,B 0,C 180,E1 5688.794,E2 5688.794} C_VEL
LIN {X 0,Y 653.282,Z 1064.951,A -85,B 0,C 180,E1 5692.325,E2 5692.325} C_VEL
LIN {X 0,Y 655.808,Z 1029.08,A -85,B 0,C 180,E1 5695.596,E2 5695.596} C_VEL
LIN {X 0,Y 658.571,Z 989.25,A -85,B 0,C 180,E1 5698.385,E2 5698.385} C_VEL
LIN {X 0,Y 661.389,Z 946.192,A -85,B 0,C 180,E1 5700.639,E2 5700.639} C_VEL
LIN {X 0,Y 663.772,Z 901.336,A -85,B 0,C 180,E1 5702.313,E2 5702.313} C_VEL
LIN {X 0,Y 665.43,Z 856.598,A -85,B 0,C 180,E1 5703.391,E2 5703.391} C_VEL
LIN {X 0,Y 665.788,Z 817.363,A -85,B 0,C 180,E1 5703.965,E2 5703.965} C_VEL
LIN {X 0,Y 648.573,Z 780.81,A -85,B 0,C 180,E1 5705.532,E2 5705.532} C_VEL
LIN {X 0,Y 648.522,Z 780.81,A -85,B 0,C 180,E1 5710.723,E2 5710.723} C_VEL
LIN {X 0,Y 648.586,Z 780.81,A -85,B 0,C 180,E1 5715.669,E2 5715.669} C_VEL
LIN {X 0,Y 648.479,Z 780.81,A -85,B 0,C 180,E1 5721.022,E2 5721.022} C_VEL
LIN {X 0,Y 648.512,Z 780.81,A -85,B 0,C 180,E1 5726.007,E2 5726.007} C_VEL
LIN {X 0,Y 648.63,Z 780.81,A -85,B 0,C 180,E1 5730.718,E2 5730.718} C_VEL
LIN {X 0,Y 648.757,Z 780.81,A -85,B 0,C 180,E1 5735.283,E2 5735.283} C_VEL
LIN {X 0,Y 648.813,Z 780.81,A -85,B 0,C 180,E1 5740.975,E2 5740.975} C_VEL
LIN {X 0,Y 648.864,Z 780.81,A -85,B 0,C 180,E1 5745.162,E2 5745.162} C_VEL
LIN {X 0,Y 648.946,Z 780.81,A -85,B 0,C 180,E1 5750.623,E2 5750.623} C_VEL
LIN {X 0,Y 649.119,Z 780.81,A -85,B 0,C 180,E1 5755.998,E2 5755.998} C_VEL
LIN {X 0,Y 649.31,Z 780.81,A -85,B 0,C 180,E1 5761.335,E2 5761.335} C_VEL
LIN {X 0,Y 649.006,Z 780.81,A -85,B 0,C 180,E1 5766.686,E2 5766.686} C_VEL
LIN {X 0,Y 648.907,Z 780.81,A -85,B 0,C 180,E1 5772.098,E2 5772.098} C_VEL
LIN {X 0,Y 648.867,Z 780.81,A -85,B 0,C 180,E1 5777.622,E2 5777.622} C_VEL
LIN {X 0,Y 648.688,Z 780.81,A -85,B 0,C 180,E1 5783.327,E2 5783.327} C_VEL
LIN {X 0,Y 648.66,Z 780.81,A -85,B 0,C 180,E1 5787.767,E2 5787.767} C_VEL
LIN {X 0,Y 648.594,Z 780.81,A -85,B 0,C 180,E1 5792.995,E2 5792.995} C_VEL
LIN {X 0,Y 648.447,Z 780.81,A -85,B 0,C 180,E1 5797.599,E2 5797.599} C_VEL
LIN {X 0,Y 648.548,Z 780.81,A -85,B 0,C 180,E1 5802.502,E2 5802.502} C_VEL
LIN {X 0,Y 648.472,Z 780.81,A -85,B 0,C 180,E1 5807.487,E2 5807.487} C_VEL
LIN {X 0,Y 648.672,Z 780.81,A -85,B 0,C 180,E1 5811.962,E2 5811.962} C_VEL
LIN {X 0,Y 665.512,Z 819.867,A -85,B 0,C 180,E1 5813.624,E2 5813.624} C_VEL
LIN {X 0,Y 663.899,Z 860.988,A -85,B 0,C 180,E1 5814.632,E2 5814.632} C_VEL
LIN {X 0,Y 661.478,Z 904.708,A -85,B 0,C 180,E1 5816.248,E2 5816.248} C_VEL
LIN {X 0,Y 658.638,Z 948.689,A -85,B 0,C 180,E1 5818.538,E2 5818.538} C_VEL
LIN {X 0,Y 655.812,Z 988.576,A -85,B 0,C 180,E1 5821.318,E2 5821.318} C_VEL
LIN {X 0,Y 653.312,Z 1023.785,A -85,B 0,C 180,E1 5824.511,E2 5824.511} C_VEL
LIN {X 0,Y 651.6,Z 1052.321,A -85,B 0,C 180,E1 5827.837,E2 5827.837} C_VEL
LIN {X 0,Y 650.266,Z 1076.169,A -85,B 0,C 180,E1 5831.402,E2 5831.402} C_VEL
LIN {X 0,Y 649.63,Z 1095.128,A -85,B 0,C 180,E1 5835.176,E2 5835.176} C_VEL
LIN {X 0,Y 649.368,Z 1107.263,A -85,B 0,C 180,E1 5838.593,E2 5838.593} C_VEL
LIN {X 0,Y 649.223,Z 1115.135,A -85,B 0,C 180,E1 5841.973,E2 5841.973} C_VEL
LIN {X 0,Y 649.19,Z 1119.265,A -85,B 0,C 180,E1 5845.997,E2 5845.997} C_VEL
LIN {X 0,Y 649.252,Z 1117.885,A -85,B 0,C 180,E1 5850.001,E2 5850.001} C_VEL
LIN {X 0,Y 649.381,Z 1110.824,A -85,B 0,C 180,E1 5854.004,E2 5854.004} C_VEL
LIN {X 0,Y 649.621,Z 1099.265,A -85,B 0,C 180,E1 5857.687,E2 5857.687} C_VEL
LIN {X 0,Y 650.175,Z 1082.392,A -85,B 0,C 180,E1 5861.395,E2 5861.395} C_VEL
LIN {X 0,Y 651.095,Z 1059.972,A -85,B 0,C 180,E1 5865.031,E2 5865.031} C_VEL
LIN {X 0,Y 652.665,Z 1033.523,A -85,B 0,C 180,E1 5868.352,E2 5868.352} C_VEL
LIN {X 0,Y 654.97,Z 1000.945,A -85,B 0,C 180,E1 5871.56,E2 5871.56} C_VEL
LIN {X 0,Y 657.625,Z 963.43,A -85,B 0,C 180,E1 5874.432,E2 5874.432} C_VEL
LIN {X 0,Y 660.475,Z 921.752,A -85,B 0,C 180,E1 5876.853,E2 5876.853} C_VEL
LIN {X 0,Y 662.799,Z 881.054,A -85,B 0,C 180,E1 5878.606,E2 5878.606} C_VEL
LIN {X 0,Y 664.791,Z 839.989,A -85,B 0,C 180,E1 5879.855,E2 5879.855} C_VEL
LIN {X 0,Y 664.938,Z 816.725,A -85,B 0,C 180,E1 5880.381,E2 5880.381} C_VEL
LIN {X 0,Y 648.661,Z 780.81,A -85,B 0,C 180,E1 5882.002,E2 5882.002} C_VEL
LIN {X 0,Y 648.442,Z 780.81,A -85,B 0,C 180,E1 5887.606,E2 5887.606} C_VEL
LIN {X 0,Y 648.552,Z 780.81,A -85,B 0,C 180,E1 5892.509,E2 5892.509} C_VEL
LIN {X 0,Y 648.454,Z 780.81,A -85,B 0,C 180,E1 5897.491,E2 5897.491} C_VEL
LIN {X 0,Y 648.457,Z 780.81,A -85,B 0,C 180,E1 5902.713,E2 5902.713} C_VEL
LIN {X 0,Y 648.489,Z 780.81,A -85,B 0,C 180,E1 5907.596,E2 5907.596} C_VEL
LIN {X 0,Y 648.725,Z 780.81,A -85,B 0,C 180,E1 5912.272,E2 5912.272} C_VEL
LIN {X 0,Y 648.716,Z 780.81,A -85,B 0,C 180,E1 5916.674,E2 5916.674} C_VEL
LIN {X 0,Y 648.862,Z 780.81,A -85,B 0,C 180,E1 5922.378,E2 5922.378} C_VEL
LIN {X 0,Y 648.913,Z 780.81,A -85,B 0,C 180,E1 5927.974,E2 5927.974} C_VEL
LIN {X 0,Y 649.095,Z 780.81,A -85,B 0,C 180,E1 5933.315,E2 5933.315} C_VEL
LIN {X 0,Y 649.127,Z 780.81,A -85,B 0,C 180,E1 5938.664,E2 5938.664} C_VEL
LIN {X 0,Y 649.064,Z 780.81,A -85,B 0,C 180,E1 5942.666,E2 5942.666} C_VEL
LIN {X 0,Y 649.015,Z 780.81,A -85,B 0,C 180,E1 5948.027,E2 5948.027} C_VEL
LIN {X 0,Y 648.894,Z 780.81,A -85,B 0,C 180,E1 5953.462,E2 5953.462} C_VEL
LIN {X 0,Y 648.849,Z 780.81,A -85,B 0,C 180,E1 5959.023,E2 5959.023} C_VEL
LIN {X 0,Y 648.736,Z 780.81,A -85,B 0,C 180,E1 5964.709,E2 5964.709} C_VEL
LIN {X 0,Y 648.663,Z 780.81,A -85,B 0,C 180,E1 5969.281,E2 5969.281} C_VEL
LIN {X 0,Y 648.592,Z 780.81,A -85,B 0,C 180,E1 5974.695,E2 5974.695} C_VEL
LIN {X 0,Y 647.311,Z 780.81,A -85,B 0,C 180,E1 5975.461,E2 5975.461} C_VEL
LIN {X 0,Y 640.628,Z 780.81,A -85,B 0,C 180,E1 5977.541,E2 5977.541} C_VEL
LIN {X 0,Y 640.546,Z 780.81,A -85,B 0,C 180,E1 5977.738,E2 5977.738} C_VEL
LIN {X 0,Y 640.512,Z 780.81,A -85,B 0,C 180,E1 5983.158,E2 5983.158} C_VEL
LIN {X 0,Y 640.516,Z 780.81,A -85,B 0,C 180,E1 5988.655,E2 5988.655} C_VEL
LIN {X 0,Y 640.648,Z 780.81,A -85,B 0,C 180,E1 5994.005,E2 5994.005} C_VEL
LIN {X 0,Y 659.476,Z 820.612,A -85,B 0,C 180,E1 5995.71,E2 5995.71} C_VEL
LIN {X 0,Y 658.401,Z 868.882,A -85,B 0,C 180,E1 5996.477,E2 5996.477} C_VEL
LIN {X 0,Y 656.423,Z 913.925,A -85,B 0,C 180,E1 5997.73,E2 5997.73} C_VEL
LIN {X 0,Y 653.61,Z 958.908,A -85,B 0,C 180,E1 5999.601,E2 5999.601} C_VEL
LIN {X 0,Y 650.631,Z 1000.408,A -85,B 0,C 180,E1 6001.995,E2 6001.995} C_VEL
LIN {X 0,Y 647.849,Z 1036.473,A -85,B 0,C 180,E1 6004.713,E2 6004.713} C_VEL
LIN {X 0,Y 645.517,Z 1067.715,A -85,B 0,C 180,E1 6007.697,E2 6007.697} C_VEL
LIN {X 0,Y 643.679,Z 1097.389,A -85,B 0,C 180,E1 6011.33,E2 6011.33} C_VEL
LIN {X 0,Y 642.467,Z 1120.359,A -85,B 0,C 180,E1 6015.005,E2 6015.005} C_VEL
LIN {X 0,Y 641.671,Z 1137.956,A -85,B 0,C 180,E1 6018.796,E2 6018.796} C_VEL
LIN {X 0,Y 641.429,Z 1150.116,A -85,B 0,C 180,E1 6022.554,E2 6022.554} C_VEL
LIN {X 0,Y 641.296,Z 1156.662,A -85,B 0,C 180,E1 6025.946,E2 6025.946} C_VEL
LIN {X 0,Y 641.29,Z 1159.5,A -85,B 0,C 180,E1 6029.999,E2 6029.999} C_VEL
LIN {X 0,Y 641.275,Z 1156.665,A -85,B 0,C 180,E1 6034.053,E2 6034.053} C_VEL
LIN {X 0,Y 641.505,Z 1150.119,A -85,B 0,C 180,E1 6037.443,E2 6037.443} C_VEL
LIN {X 0,Y 641.821,Z 1136.626,A -85,B 0,C 180,E1 6041.543,E2 6041.543} C_VEL
LIN {X 0,Y 642.606,Z 1117.876,A -85,B 0,C 180,E1 6045.437,E2 6045.437} C_VEL
LIN {X 0,Y 643.802,Z 1095.495,A -85,B 0,C 180,E1 6048.932,E2 6048.932} C_VEL
LIN {X 0,Y 645.715,Z 1064.95,A -85,B 0,C 180,E1 6052.601,E2 6052.601} C_VEL
LIN {X 0,Y 648.442,Z 1029.082,A -85,B 0,C 180,E1 6055.908,E2 6055.908} C_VEL
LIN {X 0,Y 651.491,Z 988.911,A -85,B 0,C 180,E1 6058.744,E2 6058.744} C_VEL
LIN {X 0,Y 654.52,Z 946.11,A -85,B 0,C 180,E1 6060.999,E2 6060.999} C_VEL
LIN {X 0,Y 657.001,Z 901.198,A -85,B 0,C 180,E1 6062.681,E2 6062.681} C_VEL
LIN {X 0,Y 658.778,Z 857.228,A -85,B 0,C 180,E1 6063.754,E2 6063.754} C_VEL
LIN {X 0,Y 658.977,Z 819.368,A -85,B 0,C 180,E1 6064.335,E2 6064.335} C_VEL
LIN {X 0,Y 640.62,Z 780.81,A -85,B 0,C 180,E1 6065.994,E2 6065.994} C_VEL
LIN {X 0,Y 640.626,Z 780.81,A -85,B 0,C 180,E1 6071.334,E2 6071.334} C_VEL
LIN {X 0,Y 640.601,Z 780.81,A -85,B 0,C 180,E1 6076.849,E2 6076.849} C_VEL
LIN {X 0,Y 640.584,Z 780.81,A -85,B 0,C 180,E1 6082.18,E2 6082.18} C_VEL
LIN {X 0,Y 640.583,Z 780.81,A -85,B 0,C 180,E1 6087.151,E2 6087.151} C_VEL
LIN {X 0,Y 640.76,Z 780.81,A -85,B 0,C 180,E1 6091.865,E2 6091.865} C_VEL
LIN {X 0,Y 640.826,Z 780.81,A -85,B 0,C 180,E1 6096.872,E2 6096.872} C_VEL
LIN {X 0,Y 640.915,Z 780.81,A -85,B 0,C 180,E1 6102.157,E2 6102.157} C_VEL
LIN {X 0,Y 640.874,Z 780.81,A -85,B 0,C 180,E1 6106.366,E2 6106.366} C_VEL
LIN {X 0,Y 641.115,Z 780.81,A -85,B 0,C 180,E1 6111.873,E2 6111.873} C_VEL
LIN {X 0,Y 641.291,Z 780.81,A -85,B 0,C 180,E1 6117.301,E2 6117.301} C_VEL
LIN {X 0,Y 641.168,Z 780.81,A -85,B 0,C 180,E1 6122.703,E2 6122.703} C_VEL
LIN {X 0,Y 641.097,Z 780.81,A -85,B 0,C 180,E1 6126.769,E2 6126.769} C_VEL
LIN {X 0,Y 641.021,Z 780.81,A -85,B 0,C 180,E1 6130.871,E2 6130.871} C_VEL
LIN {X 0,Y 640.993,Z 780.81,A -85,B 0,C 180,E1 6136.432,E2 6136.432} C_VEL
LIN {X 0,Y 640.876,Z 780.81,A -85,B 0,C 180,E1 6140.711,E2 6140.711} C_VEL
LIN {X 0,Y 640.758,Z 780.81,A -85,B 0,C 180,E1 6146.344,E2 6146.344} C_VEL
LIN {X 0,Y 640.648,Z 780.81,A -85,B 0,C 180,E1 6151.884,E2 6151.884} C_VEL
LIN {X 0,Y 640.546,Z 780.81,A -85,B 0,C 180,E1 6156.671,E2 6156.671} C_VEL
LIN {X 0,Y 640.571,Z 780.81,A -85,B 0,C 180,E1 6161.334,E2 6161.334} C_VEL
LIN {X 0,Y 640.586,Z 780.81,A -85,B 0,C 180,E1 6166.986,E2 6166.986} C_VEL
LIN {X 0,Y 640.742,Z 780.817,A -85,B 0,C 180,E1 6171.491,E2 6171.491} C_VEL
LIN {X 0,Y 648.979,Z 798.903,A -85,B 0,C 180,E1 6172.265,E2 6172.265} C_VEL
LIN {X 0,Y 658.845,Z 822.931,A -85,B 0,C 180,E1 6173.299,E2 6173.299} C_VEL
LIN {X 0,Y 657.062,Z 863.756,A -85,B 0,C 180,E1 6174.344,E2 6174.344} C_VEL
LIN {X 0,Y 654.5,Z 906.144,A -85,B 0,C 180,E1 6175.954,E2 6175.954} C_VEL
LIN {X 0,Y 651.49,Z 949.509,A -85,B 0,C 180,E1 6178.25,E2 6178.25} C_VEL
LIN {X 0,Y 648.399,Z 989.731,A -85,B 0,C 180,E1 6181.098,E2 6181.098} C_VEL
LIN {X 0,Y 645.691,Z 1025.533,A -85,B 0,C 180,E1 6184.414,E2 6184.414} C_VEL
LIN {X 0,Y 643.677,Z 1056.245,A -85,B 0,C 180,E1 6188.12,E2 6188.12} C_VEL
LIN {X 0,Y 642.391,Z 1079.703,A -85,B 0,C 180,E1 6191.84,E2 6191.84} C_VEL
LIN {X 0,Y 641.736,Z 1096.342,A -85,B 0,C 180,E1 6195.338,E2 6195.338} C_VEL
LIN {X 0,Y 641.459,Z 1109.094,A -85,B 0,C 180,E1 6199.138,E2 6199.138} C_VEL
LIN {X 0,Y 641.274,Z 1116.224,A -85,B 0,C 180,E1 6202.554,E2 6202.554} C_VEL
LIN {X 0,Y 641.283,Z 1119.255,A -85,B 0,C 180,E1 6205.947,E2 6205.947} C_VEL
LIN {X 0,Y 641.352,Z 1117.933,A -85,B 0,C 180,E1 6210.001,E2 6210.001} C_VEL
LIN {X 0,Y 641.481,Z 1110.911,A -85,B 0,C 180,E1 6214.053,E2 6214.053} C_VEL
LIN {X 0,Y 641.743,Z 1099.414,A -85,B 0,C 180,E1 6217.782,E2 6217.782} C_VEL
LIN {X 0,Y 642.341,Z 1082.589,A -85,B 0,C 180,E1 6221.536,E2 6221.536} C_VEL
LIN {X 0,Y 643.335,Z 1060.572,A -85,B 0,C 180,E1 6225.168,E2 6225.168} C_VEL
LIN {X 0,Y 645.085,Z 1033.881,A -85,B 0,C 180,E1 6228.576,E2 6228.576} C_VEL
LIN {X 0,Y 647.502,Z 1002.028,A -85,B 0,C 180,E1 6231.767,E2 6231.767} C_VEL
LIN {X 0,Y 650.399,Z 963.996,A -85,B 0,C 180,E1 6234.722,E2 6234.722} C_VEL
LIN {X 0,Y 653.348,Z 923.715,A -85,B 0,C 180,E1 6237.103,E2 6237.103} C_VEL
LIN {X 0,Y 655.902,Z 883.9,A -85,B 0,C 180,E1 6238.871,E2 6238.871} C_VEL
LIN {X 0,Y 658.112,Z 841.916,A -85,B 0,C 180,E1 6240.19,E2 6240.19} C_VEL
LIN {X 0,Y 658.284,Z 819.355,A -85,B 0,C 180,E1 6240.716,E2 6240.716} C_VEL
LIN {X 0,Y 640.725,Z 780.81,A -85,B 0,C 180,E1 6242.48,E2 6242.48} C_VEL
LIN {X 0,Y 640.52,Z 780.81,A -85,B 0,C 180,E1 6247.836,E2 6247.836} C_VEL
LIN {X 0,Y 640.651,Z 780.81,A -85,B 0,C 180,E1 6253.16,E2 6253.16} C_VEL
LIN {X 0,Y 640.553,Z 780.81,A -85,B 0,C 180,E1 6259.018,E2 6259.018} C_VEL
LIN {X 0,Y 640.532,Z 780.81,A -85,B 0,C 180,E1 6263.863,E2 6263.863} C_VEL
LIN {X 0,Y 640.606,Z 780.81,A -85,B 0,C 180,E1 6268.742,E2 6268.742} C_VEL
LIN {X 0,Y 640.857,Z 780.81,A -85,B 0,C 180,E1 6273.641,E2 6273.641} C_VEL
LIN {X 0,Y 640.889,Z 780.81,A -85,B 0,C 180,E1 6279.289,E2 6279.289} C_VEL
LIN {X 0,Y 640.97,Z 780.81,A -85,B 0,C 180,E1 6284.97,E2 6284.97} C_VEL
LIN {X 0,Y 641.069,Z 780.81,A -85,B 0,C 180,E1 6290.502,E2 6290.502} C_VEL
LIN {X 0,Y 641.229,Z 780.81,A -85,B 0,C 180,E1 6295.945,E2 6295.945} C_VEL
LIN {X 0,Y 641.425,Z 780.81,A -85,B 0,C 180,E1 6301.348,E2 6301.348} C_VEL
LIN {X 0,Y 641.077,Z 780.81,A -85,B 0,C 180,E1 6306.765,E2 6306.765} C_VEL
LIN {X 0,Y 641.016,Z 780.81,A -85,B 0,C 180,E1 6310.866,E2 6310.866} C_VEL
LIN {X 0,Y 641.001,Z 780.81,A -85,B 0,C 180,E1 6316.428,E2 6316.428} C_VEL
LIN {X 0,Y 640.91,Z 780.81,A -85,B 0,C 180,E1 6320.706,E2 6320.706} C_VEL
LIN {X 0,Y 640.816,Z 780.81,A -85,B 0,C 180,E1 6326.351,E2 6326.351} C_VEL
LIN {X 0,Y 640.73,Z 780.81,A -85,B 0,C 180,E1 6331.893,E2 6331.893} C_VEL
LIN {X 0,Y 640.588,Z 780.81,A -85,B 0,C 180,E1 6336.674,E2 6336.674} C_VEL
LIN {X 0,Y 640.546,Z 780.81,A -85,B 0,C 180,E1 6337.738,E2 6337.738} C_VEL
LIN {X 0,Y 638.031,Z 780.81,A -85,B 0,C 180,E1 6338.881,E2 6338.881} C_VEL
LIN {X 0,Y 632.591,Z 780.81,A -85,B 0,C 180,E1 6340.59,E2 6340.59} C_VEL
LIN {X 0,Y 632.486,Z 780.81,A -85,B 0,C 180,E1 6340.788,E2 6340.788} C_VEL
LIN {X 0,Y 632.571,Z 780.81,A -85,B 0,C 180,E1 6346.15,E2 6346.15} C_VEL
LIN {X 0,Y 632.641,Z 780.81,A -85,B 0,C 180,E1 6352.004,E2 6352.004} C_VEL
LIN {X 0,Y 632.713,Z 780.81,A -85,B 0,C 180,E1 6353.49,E2 6353.49} C_VEL
LIN {X 0,Y 645.565,Z 807.815,A -85,B 0,C 180,E1 6354.702,E2 6354.702} C_VEL
LIN {X 0,Y 653.004,Z 823.553,A -85,B 0,C 180,E1 6355.364,E2 6355.364} C_VEL
LIN {X 0,Y 651.653,Z 871.222,A -85,B 0,C 180,E1 6356.15,E2 6356.15} C_VEL
LIN {X 0,Y 649.551,Z 915.008,A -85,B 0,C 180,E1 6357.402,E2 6357.402} C_VEL
LIN {X 0,Y 646.604,Z 959.433,A -85,B 0,C 180,E1 6359.274,E2 6359.274} C_VEL
LIN {X 0,Y 643.494,Z 1000.404,A -85,B 0,C 180,E1 6361.657,E2 6361.657} C_VEL
LIN {X 0,Y 640.561,Z 1035.898,A -85,B 0,C 180,E1 6364.353,E2 6364.353} C_VEL
LIN {X 0,Y 637.993,Z 1067.964,A -85,B 0,C 180,E1 6367.448,E2 6367.448} C_VEL
LIN {X 0,Y 635.962,Z 1097.497,A -85,B 0,C 180,E1 6371.11,E2 6371.11} C_VEL
LIN {X 0,Y 634.655,Z 1120.358,A -85,B 0,C 180,E1 6374.816,E2 6374.816} C_VEL
LIN {X 0,Y 633.806,Z 1138.007,A -85,B 0,C 180,E1 6378.669,E2 6378.669} C_VEL
LIN {X 0,Y 633.55,Z 1150.116,A -85,B 0,C 180,E1 6382.461,E2 6382.461} C_VEL
LIN {X 0,Y 633.4,Z 1156.661,A -85,B 0,C 180,E1 6385.895,E2 6385.895} C_VEL
LIN {X 0,Y 633.392,Z 1159.5,A -85,B 0,C 180,E1 6389.999,E2 6389.999} C_VEL
LIN {X 0,Y 633.381,Z 1156.664,A -85,B 0,C 180,E1 6394.104,E2 6394.104} C_VEL
LIN {X 0,Y 633.621,Z 1150.119,A -85,B 0,C 180,E1 6397.536,E2 6397.536} C_VEL
LIN {X 0,Y 633.953,Z 1136.749,A -85,B 0,C 180,E1 6401.657,E2 6401.657} C_VEL
LIN {X 0,Y 634.824,Z 1117.874,A -85,B 0,C 180,E1 6405.631,E2 6405.631} C_VEL
LIN {X 0,Y 636.09,Z 1095.08,A -85,B 0,C 180,E1 6409.227,E2 6409.227} C_VEL
LIN {X 0,Y 638.116,Z 1066.243,A -85,B 0,C 180,E1 6412.744,E2 6412.744} C_VEL
LIN {X 0,Y 640.949,Z 1031.897,A -85,B 0,C 180,E1 6415.988,E2 6415.988} C_VEL
LIN {X 0,Y 643.914,Z 994.299,A -85,B 0,C 180,E1 6418.744,E2 6418.744} C_VEL
LIN {X 0,Y 646.874,Z 955.242,A -85,B 0,C 180,E1 6420.925,E2 6420.925} C_VEL
LIN {X 0,Y 649.691,Z 911.345,A -85,B 0,C 180,E1 6422.727,E2 6422.727} C_VEL
LIN {X 0,Y 651.964,Z 864.629,A -85,B 0,C 180,E1 6423.997,E2 6423.997} C_VEL
LIN {X 0,Y 652.418,Z 822.01,A -85,B 0,C 180,E1 6424.69,E2 6424.69} C_VEL
LIN {X 0,Y 632.678,Z 780.81,A -85,B 0,C 180,E1 6426.54,E2 6426.54} C_VEL
LIN {X 0,Y 632.7,Z 780.81,A -85,B 0,C 180,E1 6432.25,E2 6432.25} C_VEL
LIN {X 0,Y 632.615,Z 780.81,A -85,B 0,C 180,E1 6438.035,E2 6438.035} C_VEL
LIN {X 0,Y 632.684,Z 780.81,A -85,B 0,C 180,E1 6443.347,E2 6443.347} C_VEL
LIN {X 0,Y 632.708,Z 780.81,A -85,B 0,C 180,E1 6449.292,E2 6449.292} C_VEL
LIN {X 0,Y 632.902,Z 780.81,A -85,B 0,C 180,E1 6454.554,E2 6454.554} C_VEL
LIN {X 0,Y 632.983,Z 780.81,A -85,B 0,C 180,E1 6460.481,E2 6460.481} C_VEL
LIN {X 0,Y 633.05,Z 780.81,A -85,B 0,C 180,E1 6464.782,E2 6464.782} C_VEL
LIN {X 0,Y 633.118,Z 780.81,A -85,B 0,C 180,E1 6470.386,E2 6470.386} C_VEL
LIN {X 0,Y 633.307,Z 780.81,A -85,B 0,C 180,E1 6475.898,E2 6475.898} C_VEL
LIN {X 0,Y 633.508,Z 780.81,A -85,B 0,C 180,E1 6481.369,E2 6481.369} C_VEL
LIN {X 0,Y 633.19,Z 780.81,A -85,B 0,C 180,E1 6486.854,E2 6486.854} C_VEL
LIN {X 0,Y 633.06,Z 780.81,A -85,B 0,C 180,E1 6491.861,E2 6491.861} C_VEL
LIN {X 0,Y 633.031,Z 780.81,A -85,B 0,C 180,E1 6497.288,E2 6497.288} C_VEL
LIN {X 0,Y 632.873,Z 780.81,A -85,B 0,C 180,E1 6502.458,E2 6502.458} C_VEL
LIN {X 0,Y 632.788,Z 780.81,A -85,B 0,C 180,E1 6507.926,E2 6507.926} C_VEL
LIN {X 0,Y 632.749,Z 780.81,A -85,B 0,C 180,E1 6513.313,E2 6513.313} C_VEL
LIN {X 0,Y 632.602,Z 780.81,A -85,B 0,C 180,E1 6518.389,E2 6518.389} C_VEL
LIN {X 0,Y 632.663,Z 780.81,A -85,B 0,C 180,E1 6524.231,E2 6524.231} C_VEL
LIN {X 0,Y 632.681,Z 780.81,A -85,B 0,C 180,E1 6529.845,E2 6529.845} C_VEL
LIN {X 0,Y 632.798,Z 781.516,A -85,B 0,C 180,E1 6530.982,E2 6530.982} C_VEL
LIN {X 0,Y 652.218,Z 823.883,A -85,B 0,C 180,E1 6532.924,E2 6532.924} C_VEL
LIN {X 0,Y 650.359,Z 864.748,A -85,B 0,C 180,E1 6533.991,E2 6533.991} C_VEL
LIN {X 0,Y 647.679,Z 905.954,A -85,B 0,C 180,E1 6535.566,E2 6535.566} C_VEL
LIN {X 0,Y 644.465,Z 948.557,A -85,B 0,C 180,E1 6537.845,E2 6537.845} C_VEL
LIN {X 0,Y 641.209,Z 988.378,A -85,B 0,C 180,E1 6540.674,E2 6540.674} C_VEL
LIN {X 0,Y 638.348,Z 1023.163,A -85,B 0,C 180,E1 6543.89,E2 6543.89} C_VEL
LIN {X 0,Y 636.298,Z 1051.892,A -85,B 0,C 180,E1 6547.301,E2 6547.301} C_VEL
LIN {X 0,Y 634.808,Z 1075.521,A -85,B 0,C 180,E1 6550.895,E2 6550.895} C_VEL
LIN {X 0,Y 633.961,Z 1094.783,A -85,B 0,C 180,E1 6554.8,E2 6554.8} C_VEL
LIN {X 0,Y 633.62,Z 1107.381,A -85,B 0,C 180,E1 6558.426,E2 6558.426} C_VEL
LIN {X 0,Y 633.404,Z 1116.176,A -85,B 0,C 180,E1 6562.461,E2 6562.461} C_VEL
LIN {X 0,Y 633.375,Z 1119.245,A -85,B 0,C 180,E1 6565.896,E2 6565.896} C_VEL
LIN {X 0,Y 633.452,Z 1117.976,A -85,B 0,C 180,E1 6570.001,E2 6570.001} C_VEL
LIN {X 0,Y 633.604,Z 1110.997,A -85,B 0,C 180,E1 6574.104,E2 6574.104} C_VEL
LIN {X 0,Y 633.861,Z 1099.563,A -85,B 0,C 180,E1 6577.88,E2 6577.88} C_VEL
LIN {X 0,Y 634.527,Z 1082.787,A -85,B 0,C 180,E1 6581.68,E2 6581.68} C_VEL
LIN {X 0,Y 635.68,Z 1060.033,A -85,B 0,C 180,E1 6585.475,E2 6585.475} C_VEL
LIN {X 0,Y 637.643,Z 1032.602,A -85,B 0,C 180,E1 6588.987,E2 6588.987} C_VEL
LIN {X 0,Y 640.2,Z 1000.691,A -85,B 0,C 180,E1 6592.19,E2 6592.19} C_VEL
LIN {X 0,Y 643.324,Z 963.038,A -85,B 0,C 180,E1 6595.125,E2 6595.125} C_VEL
LIN {X 0,Y 646.587,Z 921.873,A -85,B 0,C 180,E1 6597.568,E2 6597.568} C_VEL
LIN {X 0,Y 649.325,Z 881.252,A -85,B 0,C 180,E1 6599.352,E2 6599.352} C_VEL
LIN {X 0,Y 651.572,Z 840.399,A -85,B 0,C 180,E1 6600.614,E2 6600.614} C_VEL
LIN {X 0,Y 651.844,Z 822.532,A -85,B 0,C 180,E1 6601.036,E2 6601.036} C_VEL
LIN {X 0,Y 632.787,Z 780.81,A -85,B 0,C 180,E1 6602.983,E2 6602.983} C_VEL
LIN {X 0,Y 632.599,Z 780.81,A -85,B 0,C 180,E1 6608.395,E2 6608.395} C_VEL
LIN {X 0,Y 632.668,Z 780.81,A -85,B 0,C 180,E1 6614.238,E2 6614.238} C_VEL
LIN {X 0,Y 632.623,Z 780.81,A -85,B 0,C 180,E1 6619.852,E2 6619.852} C_VEL
LIN {X 0,Y 632.61,Z 780.81,A -85,B 0,C 180,E1 6625.025,E2 6625.025} C_VEL
LIN {X 0,Y 632.732,Z 780.81,A -85,B 0,C 180,E1 6629.902,E2 6629.902} C_VEL
LIN {X 0,Y 632.886,Z 780.81,A -85,B 0,C 180,E1 6635.137,E2 6635.137} C_VEL
LIN {X 0,Y 633.001,Z 780.81,A -85,B 0,C 180,E1 6640.477,E2 6640.477} C_VEL
LIN {X 0,Y 633.051,Z 780.81,A -85,B 0,C 180,E1 6644.778,E2 6644.778} C_VEL
LIN {X 0,Y 633.154,Z 780.81,A -85,B 0,C 180,E1 6650.382,E2 6650.382} C_VEL
LIN {X 0,Y 633.328,Z 780.81,A -85,B 0,C 180,E1 6655.894,E2 6655.894} C_VEL
LIN {X 0,Y 633.529,Z 780.81,A -85,B 0,C 180,E1 6661.364,E2 6661.364} C_VEL
LIN {X 0,Y 633.172,Z 780.81,A -85,B 0,C 180,E1 6666.85,E2 6666.85} C_VEL
LIN {X 0,Y 633.091,Z 780.81,A -85,B 0,C 180,E1 6671.867,E2 6671.867} C_VEL
LIN {X 0,Y 633.048,Z 780.81,A -85,B 0,C 180,E1 6677.288,E2 6677.288} C_VEL
LIN {X 0,Y 632.92,Z 780.81,A -85,B 0,C 180,E1 6682.451,E2 6682.451} C_VEL
LIN {X 0,Y 632.86,Z 780.81,A -85,B 0,C 180,E1 6687.935,E2 6687.935} C_VEL
LIN {X 0,Y 632.824,Z 780.81,A -85,B 0,C 180,E1 6693.304,E2 6693.304} C_VEL
LIN {X 0,Y 632.617,Z 780.81,A -85,B 0,C 180,E1 6698.382,E2 6698.382} C_VEL
LIN {X 0,Y 632.486,Z 780.81,A -85,B 0,C 180,E1 6700.788,E2 6700.788} C_VEL
LIN {X 0,Y 628.516,Z 780.81,A -85,B 0,C 180,E1 6702.339,E2 6702.339} C_VEL
LIN {X 0,Y 624.581,Z 780.81,A -85,B 0,C 180,E1 6703.91,E2 6703.91} C_VEL
LIN {X 0,Y 624.597,Z 780.81,A -85,B 0,C 180,E1 6709.214,E2 6709.214} C_VEL
LIN {X 0,Y 624.749,Z 780.958,A -85,B 0,C 180,E1 6712.983,E2 6712.983} C_VEL
LIN {X 0,Y 646.358,Z 825.74,A -85,B 0,C 180,E1 6714.989,E2 6714.989} C_VEL
LIN {X 0,Y 644.998,Z 872.247,A -85,B 0,C 180,E1 6715.786,E2 6715.786} C_VEL
LIN {X 0,Y 642.787,Z 914.942,A -85,B 0,C 180,E1 6717.024,E2 6717.024} C_VEL
LIN {X 0,Y 639.629,Z 959.602,A -85,B 0,C 180,E1 6718.926,E2 6718.926} C_VEL
LIN {X 0,Y 636.137,Z 1003.022,A -85,B 0,C 180,E1 6721.489,E2 6721.489} C_VEL
LIN {X 0,Y 632.877,Z 1039.994,A -85,B 0,C 180,E1 6724.39,E2 6724.39} C_VEL
LIN {X 0,Y 630.065,Z 1072.01,A -85,B 0,C 180,E1 6727.62,E2 6727.62} C_VEL
LIN {X 0,Y 628.178,Z 1098.705,A -85,B 0,C 180,E1 6731.049,E2 6731.049} C_VEL
LIN {X 0,Y 626.739,Z 1122.249,A -85,B 0,C 180,E1 6734.977,E2 6734.977} C_VEL
LIN {X 0,Y 625.887,Z 1139.289,A -85,B 0,C 180,E1 6738.863,E2 6738.863} C_VEL
LIN {X 0,Y 625.667,Z 1150.337,A -85,B 0,C 180,E1 6742.465,E2 6742.465} C_VEL
LIN {X 0,Y 625.506,Z 1156.661,A -85,B 0,C 180,E1 6745.843,E2 6745.843} C_VEL
LIN {X 0,Y 625.493,Z 1159.5,A -85,B 0,C 180,E1 6749.999,E2 6749.999} C_VEL
LIN {X 0,Y 625.487,Z 1156.664,A -85,B 0,C 180,E1 6754.155,E2 6754.155} C_VEL
LIN {X 0,Y 625.738,Z 1150.295,A -85,B 0,C 180,E1 6757.553,E2 6757.553} C_VEL
LIN {X 0,Y 626.079,Z 1136.99,A -85,B 0,C 180,E1 6761.742,E2 6761.742} C_VEL
LIN {X 0,Y 626.992,Z 1118.613,A -85,B 0,C 180,E1 6765.695,E2 6765.695} C_VEL
LIN {X 0,Y 628.351,Z 1094.946,A -85,B 0,C 180,E1 6769.491,E2 6769.491} C_VEL
LIN {X 0,Y 630.735,Z 1064.941,A -85,B 0,C 180,E1 6773.169,E2 6773.169} C_VEL
LIN {X 0,Y 633.856,Z 1029.53,A -85,B 0,C 180,E1 6776.513,E2 6776.513} C_VEL
LIN {X 0,Y 637.152,Z 990.44,A -85,B 0,C 180,E1 6779.333,E2 6779.333} C_VEL
LIN {X 0,Y 640.499,Z 948.494,A -85,B 0,C 180,E1 6781.601,E2 6781.601} C_VEL
LIN {X 0,Y 643.269,Z 906.316,A -85,B 0,C 180,E1 6783.264,E2 6783.264} C_VEL
LIN {X 0,Y 645.429,Z 862.896,A -85,B 0,C 180,E1 6784.42,E2 6784.42} C_VEL
LIN {X 0,Y 645.916,Z 824.683,A -85,B 0,C 180,E1 6785.051,E2 6785.051} C_VEL
LIN {X 0,Y 624.732,Z 780.81,A -85,B 0,C 180,E1 6787.057,E2 6787.057} C_VEL
LIN {X 0,Y 624.781,Z 780.81,A -85,B 0,C 180,E1 6792.625,E2 6792.625} C_VEL
LIN {X 0,Y 624.702,Z 780.81,A -85,B 0,C 180,E1 6797.379,E2 6797.379} C_VEL
LIN {X 0,Y 624.759,Z 780.81,A -85,B 0,C 180,E1 6802.954,E2 6802.954} C_VEL
LIN {X 0,Y 624.742,Z 780.81,A -85,B 0,C 180,E1 6807.859,E2 6807.859} C_VEL
LIN {X 0,Y 624.923,Z 780.81,A -85,B 0,C 180,E1 6813.466,E2 6813.466} C_VEL
LIN {X 0,Y 625.022,Z 780.81,A -85,B 0,C 180,E1 6818.743,E2 6818.743} C_VEL
LIN {X 0,Y 625.147,Z 780.81,A -85,B 0,C 180,E1 6824.585,E2 6824.585} C_VEL
LIN {X 0,Y 625.217,Z 780.81,A -85,B 0,C 180,E1 6830.263,E2 6830.263} C_VEL
LIN {X 0,Y 625.395,Z 780.81,A -85,B 0,C 180,E1 6835.846,E2 6835.846} C_VEL
LIN {X 0,Y 625.601,Z 780.81,A -85,B 0,C 180,E1 6841.386,E2 6841.386} C_VEL
LIN {X 0,Y 625.283,Z 780.81,A -85,B 0,C 180,E1 6846.941,E2 6846.941} C_VEL
LIN {X 0,Y 625.19,Z 780.81,A -85,B 0,C 180,E1 6851.149,E2 6851.149} C_VEL
LIN {X 0,Y 625.142,Z 780.81,A -85,B 0,C 180,E1 6856.861,E2 6856.861} C_VEL
LIN {X 0,Y 625.018,Z 780.81,A -85,B 0,C 180,E1 6861.262,E2 6861.262} C_VEL
LIN {X 0,Y 624.866,Z 780.81,A -85,B 0,C 180,E1 6866.524,E2 6866.524} C_VEL
LIN {X 0,Y 624.838,Z 780.81,A -85,B 0,C 180,E1 6872.175,E2 6872.175} C_VEL
LIN {X 0,Y 624.732,Z 780.81,A -85,B 0,C 180,E1 6877.203,E2 6877.203} C_VEL
LIN {X 0,Y 624.724,Z 780.81,A -85,B 0,C 180,E1 6882.625,E2 6882.625} C_VEL
LIN {X 0,Y 624.695,Z 780.81,A -85,B 0,C 180,E1 6887.368,E2 6887.368} C_VEL
LIN {X 0,Y 624.842,Z 780.81,A -85,B 0,C 180,E1 6890.403,E2 6890.403} C_VEL
LIN {X 0,Y 645.6,Z 826.248,A -85,B 0,C 180,E1 6892.571,E2 6892.571} C_VEL
LIN {X 0,Y 643.377,Z 871.027,A -85,B 0,C 180,E1 6893.804,E2 6893.804} C_VEL
LIN {X 0,Y 640.482,Z 911.113,A -85,B 0,C 180,E1 6895.428,E2 6895.428} C_VEL
LIN {X 0,Y 637.233,Z 951.288,A -85,B 0,C 180,E1 6897.654,E2 6897.654} C_VEL
LIN {X 0,Y 633.82,Z 989.573,A -85,B 0,C 180,E1 6900.444,E2 6900.444} C_VEL
LIN {X 0,Y 630.717,Z 1024.935,A -85,B 0,C 180,E1 6903.783,E2 6903.783} C_VEL
LIN {X 0,Y 628.456,Z 1054.279,A -85,B 0,C 180,E1 6907.375,E2 6907.375} C_VEL
LIN {X 0,Y 626.925,Z 1077.276,A -85,B 0,C 180,E1 6911.011,E2 6911.011} C_VEL
LIN {X 0,Y 626.078,Z 1095.667,A -85,B 0,C 180,E1 6914.865,E2 6914.865} C_VEL
LIN {X 0,Y 625.706,Z 1108.878,A -85,B 0,C 180,E1 6918.861,E2 6918.861} C_VEL
LIN {X 0,Y 625.521,Z 1115.551,A -85,B 0,C 180,E1 6922.024,E2 6922.024} C_VEL
LIN {X 0,Y 625.468,Z 1119.235,A -85,B 0,C 180,E1 6925.844,E2 6925.844} C_VEL
LIN {X 0,Y 625.551,Z 1118.012,A -85,B 0,C 180,E1 6930.001,E2 6930.001} C_VEL
LIN {X 0,Y 625.703,Z 1111.084,A -85,B 0,C 180,E1 6934.156,E2 6934.156} C_VEL
LIN {X 0,Y 625.977,Z 1099.299,A -85,B 0,C 180,E1 6938.088,E2 6938.088} C_VEL
LIN {X 0,Y 626.788,Z 1081.2,A -85,B 0,C 180,E1 6942.179,E2 6942.179} C_VEL
LIN {X 0,Y 628.231,Z 1056.746,A -85,B 0,C 180,E1 6946.199,E2 6946.199} C_VEL
LIN {X 0,Y 630.616,Z 1026.396,A -85,B 0,C 180,E1 6949.967,E2 6949.967} C_VEL
LIN {X 0,Y 633.67,Z 991.161,A -85,B 0,C 180,E1 6953.33,E2 6953.33} C_VEL
LIN {X 0,Y 637.034,Z 953.165,A -85,B 0,C 180,E1 6956.133,E2 6956.133} C_VEL
LIN {X 0,Y 640.339,Z 913.955,A -85,B 0,C 180,E1 6958.339,E2 6958.339} C_VEL
LIN {X 0,Y 643.253,Z 872.761,A -85,B 0,C 180,E1 6960.049,E2 6960.049} C_VEL
LIN {X 0,Y 645.595,Z 828.054,A -85,B 0,C 180,E1 6961.292,E2 6961.292} C_VEL
LIN {X 0,Y 641.388,Z 816.107,A -85,B 0,C 180,E1 6961.814,E2 6961.814} C_VEL
LIN {X 0,Y 624.816,Z 780.81,A -85,B 0,C 180,E1 6963.5,E2 6963.5} C_VEL
LIN {X 0,Y 624.627,Z 780.81,A -85,B 0,C 180,E1 6969.281,E2 6969.281} C_VEL
LIN {X 0,Y 624.723,Z 780.81,A -85,B 0,C 180,E1 6974.546,E2 6974.546} C_VEL
LIN {X 0,Y 624.635,Z 780.81,A -85,B 0,C 180,E1 6979.224,E2 6979.224} C_VEL
LIN {X 0,Y 624.698,Z 780.81,A -85,B 0,C 180,E1 6984.516,E2 6984.516} C_VEL
LIN {X 0,Y 624.803,Z 780.81,A -85,B 0,C 180,E1 6989.48,E2 6989.48} C_VEL
LIN {X 0,Y 624.955,Z 780.81,A -85,B 0,C 180,E1 6994.203,E2 6994.203} C_VEL
LIN {X 0,Y 625.035,Z 780.81,A -85,B 0,C 180,E1 6998.739,E2 6998.739} C_VEL
LIN {X 0,Y 625.142,Z 780.81,A -85,B 0,C 180,E1 7003.139,E2 7003.139} C_VEL
LIN {X 0,Y 625.213,Z 780.81,A -85,B 0,C 180,E1 7008.851,E2 7008.851} C_VEL
LIN {X 0,Y 625.35,Z 780.81,A -85,B 0,C 180,E1 7013.137,E2 7013.137} C_VEL
LIN {X 0,Y 625.447,Z 780.81,A -85,B 0,C 180,E1 7018.614,E2 7018.614} C_VEL
LIN {X 0,Y 625.367,Z 780.81,A -85,B 0,C 180,E1 7022.767,E2 7022.767} C_VEL
LIN {X 0,Y 625.314,Z 780.81,A -85,B 0,C 180,E1 7028.333,E2 7028.333} C_VEL
LIN {X 0,Y 625.162,Z 780.81,A -85,B 0,C 180,E1 7033.983,E2 7033.983} C_VEL
LIN {X 0,Y 625.134,Z 780.81,A -85,B 0,C 180,E1 7039.483,E2 7039.483} C_VEL
LIN {X 0,Y 624.946,Z 780.81,A -85,B 0,C 180,E1 7044.264,E2 7044.264} C_VEL
LIN {X 0,Y 624.858,Z 780.81,A -85,B 0,C 180,E1 7049.471,E2 7049.471} C_VEL
LIN {X 0,Y 624.803,Z 780.81,A -85,B 0,C 180,E1 7054.683,E2 7054.683} C_VEL
LIN {X 0,Y 624.617,Z 780.81,A -85,B 0,C 180,E1 7059.27,E2 7059.27} C_VEL
LIN {X 0,Y 624.581,Z 780.81,A -85,B 0,C 180,E1 7063.91,E2 7063.91} C_VEL
LIN {X 0,Y 620.647,Z 780.81,A -85,B 0,C 180,E1 7065.475,E2 7065.475} C_VEL
LIN {X 0,Y 616.739,Z 780.81,A -85,B 0,C 180,E1 7067.061,E2 7067.061} C_VEL
LIN {X 0,Y 616.777,Z 780.837,A -85,B 0,C 180,E1 7072.438,E2 7072.438} C_VEL
LIN {X 0,Y 623.123,Z 794.556,A -85,B 0,C 180,E1 7073.064,E2 7073.064} C_VEL
LIN {X 0,Y 639.971,Z 828.535,A -85,B 0,C 180,E1 7074.629,E2 7074.629} C_VEL
LIN {X 0,Y 638.256,Z 875.725,A -85,B 0,C 180,E1 7075.472,E2 7075.472} C_VEL
LIN {X 0,Y 635.908,Z 917.015,A -85,B 0,C 180,E1 7076.72,E2 7076.72} C_VEL
LIN {X 0,Y 632.637,Z 959.781,A -85,B 0,C 180,E1 7078.57,E2 7078.57} C_VEL
LIN {X 0,Y 628.998,Z 1002.734,A -85,B 0,C 180,E1 7081.135,E2 7081.135} C_VEL
LIN {X 0,Y 625.406,Z 1041.711,A -85,B 0,C 180,E1 7084.219,E2 7084.219} C_VEL
LIN {X 0,Y 622.253,Z 1075.532,A -85,B 0,C 180,E1 7087.739,E2 7087.739} C_VEL
LIN {X 0,Y 620.093,Z 1103.502,A -85,B 0,C 180,E1 7091.53,E2 7091.53} C_VEL
LIN {X 0,Y 618.805,Z 1124.182,A -85,B 0,C 180,E1 7095.182,E2 7095.182} C_VEL
LIN {X 0,Y 617.972,Z 1140.623,A -85,B 0,C 180,E1 7099.075,E2 7099.075} C_VEL
LIN {X 0,Y 617.722,Z 1151.676,A -85,B 0,C 180,E1 7102.974,E2 7102.974} C_VEL
LIN {X 0,Y 617.611,Z 1156.661,A -85,B 0,C 180,E1 7105.79,E2 7105.79} C_VEL
LIN {X 0,Y 617.602,Z 1159.5,A -85,B 0,C 180,E1 7109.999,E2 7109.999} C_VEL
LIN {X 0,Y 617.593,Z 1156.663,A -85,B 0,C 180,E1 7114.209,E2 7114.209} C_VEL
LIN {X 0,Y 617.873,Z 1149.189,A -85,B 0,C 180,E1 7118.082,E2 7118.082} C_VEL
LIN {X 0,Y 618.322,Z 1135.245,A -85,B 0,C 180,E1 7122.356,E2 7122.356} C_VEL
LIN {X 0,Y 619.249,Z 1116.47,A -85,B 0,C 180,E1 7126.297,E2 7126.297} C_VEL
LIN {X 0,Y 620.758,Z 1093.62,A -85,B 0,C 180,E1 7129.925,E2 7129.925} C_VEL
LIN {X 0,Y 623.224,Z 1065.611,A -85,B 0,C 180,E1 7133.392,E2 7133.392} C_VEL
LIN {X 0,Y 626.426,Z 1030.967,A -85,B 0,C 180,E1 7136.716,E2 7136.716} C_VEL
LIN {X 0,Y 629.858,Z 992.242,A -85,B 0,C 180,E1 7139.558,E2 7139.558} C_VEL
LIN {X 0,Y 633.307,Z 952.063,A -85,B 0,C 180,E1 7141.798,E2 7141.798} C_VEL
LIN {X 0,Y 636.344,Z 909.812,A -85,B 0,C 180,E1 7143.537,E2 7143.537} C_VEL
LIN {X 0,Y 638.879,Z 862.651,A -85,B 0,C 180,E1 7144.822,E2 7144.822} C_VEL
LIN {X 0,Y 639.355,Z 827.245,A -85,B 0,C 180,E1 7145.426,E2 7145.426} C_VEL
LIN {X 0,Y 616.764,Z 780.81,A -85,B 0,C 180,E1 7147.626,E2 7147.626} C_VEL
LIN {X 0,Y 616.899,Z 780.81,A -85,B 0,C 180,E1 7153.303,E2 7153.303} C_VEL
LIN {X 0,Y 616.784,Z 780.81,A -85,B 0,C 180,E1 7158.598,E2 7158.598} C_VEL
LIN {X 0,Y 616.794,Z 780.81,A -85,B 0,C 180,E1 7163.996,E2 7163.996} C_VEL
LIN {X 0,Y 616.845,Z 780.81,A -85,B 0,C 180,E1 7169.048,E2 7169.048} C_VEL
LIN {X 0,Y 617.052,Z 780.81,A -85,B 0,C 180,E1 7173.852,E2 7173.852} C_VEL
LIN {X 0,Y 617.1,Z 780.81,A -85,B 0,C 180,E1 7178.513,E2 7178.513} C_VEL
LIN {X 0,Y 617.19,Z 780.81,A -85,B 0,C 180,E1 7182.919,E2 7182.919} C_VEL
LIN {X 0,Y 617.257,Z 780.81,A -85,B 0,C 180,E1 7188.71,E2 7188.71} C_VEL
LIN {X 0,Y 617.422,Z 780.81,A -85,B 0,C 180,E1 7192.974,E2 7192.974} C_VEL
LIN {X 0,Y 617.503,Z 780.81,A -85,B 0,C 180,E1 7198.6,E2 7198.6} C_VEL
LIN {X 0,Y 617.469,Z 780.81,A -85,B 0,C 180,E1 7202.807,E2 7202.807} C_VEL
LIN {X 0,Y 617.428,Z 780.81,A -85,B 0,C 180,E1 7208.445,E2 7208.445} C_VEL
LIN {X 0,Y 617.25,Z 780.81,A -85,B 0,C 180,E1 7214.17,E2 7214.17} C_VEL
LIN {X 0,Y 617.166,Z 780.81,A -85,B 0,C 180,E1 7218.559,E2 7218.559} C_VEL
LIN {X 0,Y 617.008,Z 780.81,A -85,B 0,C 180,E1 7223.068,E2 7223.068} C_VEL
LIN {X 0,Y 616.925,Z 780.81,A -85,B 0,C 180,E1 7228.143,E2 7228.143} C_VEL
LIN {X 0,Y 616.876,Z 780.81,A -85,B 0,C 180,E1 7233.607,E2 7233.607} C_VEL
LIN {X 0,Y 616.707,Z 780.81,A -85,B 0,C 180,E1 7239.569,E2 7239.569} C_VEL
LIN {X 0,Y 616.812,Z 780.81,A -85,B 0,C 180,E1 7244.729,E2 7244.729} C_VEL
LIN {X 0,Y 616.896,Z 780.81,A -85,B 0,C 180,E1 7249.863,E2 7249.863} C_VEL
LIN {X 0,Y 621.468,Z 790.913,A -85,B 0,C 180,E1 7250.336,E2 7250.336} C_VEL
LIN {X 0,Y 638.948,Z 828.674,A -85,B 0,C 180,E1 7252.217,E2 7252.217} C_VEL
LIN {X 0,Y 636.623,Z 873.324,A -85,B 0,C 180,E1 7253.48,E2 7253.48} C_VEL
LIN {X 0,Y 633.439,Z 915.198,A -85,B 0,C 180,E1 7255.239,E2 7255.239} C_VEL
LIN {X 0,Y 630.04,Z 953.77,A -85,B 0,C 180,E1 7257.443,E2 7257.443} C_VEL
LIN {X 0,Y 626.394,Z 991.45,A -85,B 0,C 180,E1 7260.267,E2 7260.267} C_VEL
LIN {X 0,Y 623.139,Z 1025.993,A -85,B 0,C 180,E1 7263.603,E2 7263.603} C_VEL
LIN {X 0,Y 620.63,Z 1056.918,A -85,B 0,C 180,E1 7267.492,E2 7267.492} C_VEL
LIN {X 0,Y 618.94,Z 1081,A -85,B 0,C 180,E1 7271.496,E2 7271.496} C_VEL
LIN {X 0,Y 618.118,Z 1097.942,A -85,B 0,C 180,E1 7275.315,E2 7275.315} C_VEL
LIN {X 0,Y 617.818,Z 1108.769,A -85,B 0,C 180,E1 7278.717,E2 7278.717} C_VEL
LIN {X 0,Y 617.611,Z 1115.789,A -85,B 0,C 180,E1 7282.1,E2 7282.1} C_VEL
LIN {X 0,Y 617.56,Z 1119.226,A -85,B 0,C 180,E1 7285.791,E2 7285.791} C_VEL
LIN {X 0,Y 617.658,Z 1118.042,A -85,B 0,C 180,E1 7290.001,E2 7290.001} C_VEL
LIN {X 0,Y 617.817,Z 1111.171,A -85,B 0,C 180,E1 7294.209,E2 7294.209} C_VEL
LIN {X 0,Y 618.098,Z 1099.448,A -85,B 0,C 180,E1 7298.192,E2 7298.192} C_VEL
LIN {X 0,Y 618.969,Z 1081.39,A -85,B 0,C 180,E1 7302.34,E2 7302.34} C_VEL
LIN {X 0,Y 620.595,Z 1056.542,A -85,B 0,C 180,E1 7306.476,E2 7306.476} C_VEL
LIN {X 0,Y 623.21,Z 1025.55,A -85,B 0,C 180,E1 7310.355,E2 7310.355} C_VEL
LIN {X 0,Y 626.687,Z 988.682,A -85,B 0,C 180,E1 7313.878,E2 7313.878} C_VEL
LIN {X 0,Y 630.369,Z 950.107,A -85,B 0,C 180,E1 7316.711,E2 7316.711} C_VEL
LIN {X 0,Y 634.033,Z 907.33,A -85,B 0,C 180,E1 7319.054,E2 7319.054} C_VEL
LIN {X 0,Y 637.09,Z 864.442,A -85,B 0,C 180,E1 7320.726,E2 7320.726} C_VEL
LIN {X 0,Y 638.511,Z 827.26,A -85,B 0,C 180,E1 7321.756,E2 7321.756} C_VEL
LIN {X 0,Y 618.456,Z 785.552,A -85,B 0,C 180,E1 7323.836,E2 7323.836} C_VEL
LIN {X 0,Y 616.868,Z 780.81,A -85,B 0,C 180,E1 7324.055,E2 7324.055} C_VEL
LIN {X 0,Y 616.711,Z 780.81,A -85,B 0,C 180,E1 7329.575,E2 7329.575} C_VEL
LIN {X 0,Y 616.811,Z 780.81,A -85,B 0,C 180,E1 7334.734,E2 7334.734} C_VEL
LIN {X 0,Y 616.731,Z 780.81,A -85,B 0,C 180,E1 7340.433,E2 7340.433} C_VEL
LIN {X 0,Y 616.762,Z 780.81,A -85,B 0,C 180,E1 7345.705,E2 7345.705} C_VEL
LIN {X 0,Y 616.961,Z 780.81,A -85,B 0,C 180,E1 7350.672,E2 7350.672} C_VEL
LIN {X 0,Y 617.016,Z 780.81,A -85,B 0,C 180,E1 7355.398,E2 7355.398} C_VEL
LIN {X 0,Y 617.127,Z 780.81,A -85,B 0,C 180,E1 7359.953,E2 7359.953} C_VEL
LIN {X 0,Y 617.207,Z 780.81,A -85,B 0,C 180,E1 7364.377,E2 7364.377} C_VEL
LIN {X 0,Y 617.333,Z 780.81,A -85,B 0,C 180,E1 7370.133,E2 7370.133} C_VEL
LIN {X 0,Y 617.505,Z 780.81,A -85,B 0,C 180,E1 7375.789,E2 7375.789} C_VEL
LIN {X 0,Y 617.713,Z 780.81,A -85,B 0,C 180,E1 7381.399,E2 7381.399} C_VEL
LIN {X 0,Y 617.367,Z 780.81,A -85,B 0,C 180,E1 7387.026,E2 7387.026} C_VEL
LIN {X 0,Y 617.277,Z 780.81,A -85,B 0,C 180,E1 7392.723,E2 7392.723} C_VEL
LIN {X 0,Y 617.2,Z 780.81,A -85,B 0,C 180,E1 7397.281,E2 7397.281} C_VEL
LIN {X 0,Y 617.114,Z 780.81,A -85,B 0,C 180,E1 7401.543,E2 7401.543} C_VEL
LIN {X 0,Y 617.035,Z 780.81,A -85,B 0,C 180,E1 7406.149,E2 7406.149} C_VEL
LIN {X 0,Y 616.946,Z 780.81,A -85,B 0,C 180,E1 7410.988,E2 7410.988} C_VEL
LIN {X 0,Y 616.831,Z 780.81,A -85,B 0,C 180,E1 7416.056,E2 7416.056} C_VEL
LIN {X 0,Y 616.719,Z 780.81,A -85,B 0,C 180,E1 7421.408,E2 7421.408} C_VEL
LIN {X 0,Y 616.739,Z 780.81,A -85,B 0,C 180,E1 7427.061,E2 7427.061} C_VEL
LIN {X 0,Y 614.217,Z 780.81,A -85,B 0,C 180,E1 7428.252,E2 7428.252} C_VEL
LIN {X 0,Y 608.877,Z 780.81,A -85,B 0,C 180,E1 7430.033,E2 7430.033} C_VEL
LIN {X 0,Y 608.797,Z 780.81,A -85,B 0,C 180,E1 7430.239,E2 7430.239} C_VEL
LIN {X 0,Y 608.859,Z 781.478,A -85,B 0,C 180,E1 7431.893,E2 7431.893} C_VEL
LIN {X 0,Y 633.506,Z 831.308,A -85,B 0,C 180,E1 7434.257,E2 7434.257} C_VEL
LIN {X 0,Y 631.63,Z 877.53,A -85,B 0,C 180,E1 7435.112,E2 7435.112} C_VEL
LIN {X 0,Y 628.96,Z 920.298,A -85,B 0,C 180,E1 7436.455,E2 7436.455} C_VEL
LIN {X 0,Y 625.549,Z 961.711,A -85,B 0,C 180,E1 7438.304,E2 7438.304} C_VEL
LIN {X 0,Y 621.809,Z 1003.105,A -85,B 0,C 180,E1 7440.819,E2 7440.819} C_VEL
LIN {X 0,Y 618.063,Z 1041.476,A -85,B 0,C 180,E1 7443.89,E2 7443.89} C_VEL
LIN {X 0,Y 614.891,Z 1073.521,A -85,B 0,C 180,E1 7447.218,E2 7447.218} C_VEL
LIN {X 0,Y 612.726,Z 1099.901,A -85,B 0,C 180,E1 7450.739,E2 7450.739} C_VEL
LIN {X 0,Y 611.116,Z 1122.901,A -85,B 0,C 180,E1 7454.72,E2 7454.72} C_VEL
LIN {X 0,Y 610.12,Z 1140.623,A -85,B 0,C 180,E1 7458.933,E2 7458.933} C_VEL
LIN {X 0,Y 609.833,Z 1151.676,A -85,B 0,C 180,E1 7462.882,E2 7462.882} C_VEL
LIN {X 0,Y 609.717,Z 1156.66,A -85,B 0,C 180,E1 7465.735,E2 7465.735} C_VEL
LIN {X 0,Y 609.703,Z 1159.5,A -85,B 0,C 180,E1 7469.999,E2 7469.999} C_VEL
LIN {X 0,Y 609.7,Z 1156.663,A -85,B 0,C 180,E1 7474.263,E2 7474.263} C_VEL
LIN {X 0,Y 609.965,Z 1150.175,A -85,B 0,C 180,E1 7477.805,E2 7477.805} C_VEL
LIN {X 0,Y 610.384,Z 1137.544,A -85,B 0,C 180,E1 7481.898,E2 7481.898} C_VEL
LIN {X 0,Y 611.358,Z 1120.358,A -85,B 0,C 180,E1 7485.776,E2 7485.776} C_VEL
LIN {X 0,Y 612.947,Z 1096.265,A -85,B 0,C 180,E1 7489.814,E2 7489.814} C_VEL
LIN {X 0,Y 615.754,Z 1065.61,A -85,B 0,C 180,E1 7493.693,E2 7493.693} C_VEL
LIN {X 0,Y 619.153,Z 1030.667,A -85,B 0,C 180,E1 7497.055,E2 7497.055} C_VEL
LIN {X 0,Y 622.822,Z 991.943,A -85,B 0,C 180,E1 7499.926,E2 7499.926} C_VEL
LIN {X 0,Y 626.476,Z 951.567,A -85,B 0,C 180,E1 7502.197,E2 7502.197} C_VEL
LIN {X 0,Y 629.678,Z 909.51,A -85,B 0,C 180,E1 7503.94,E2 7503.94} C_VEL
LIN {X 0,Y 632.318,Z 864.045,A -85,B 0,C 180,E1 7505.198,E2 7505.198} C_VEL
LIN {X 0,Y 632.814,Z 829.767,A -85,B 0,C 180,E1 7505.809,E2 7505.809} C_VEL
LIN {X 0,Y 609.931,Z 784.792,A -85,B 0,C 180,E1 7508.052,E2 7508.052} C_VEL
LIN {X 0,Y 608.85,Z 780.81,A -85,B 0,C 180,E1 7508.23,E2 7508.23} C_VEL
LIN {X 0,Y 608.945,Z 780.81,A -85,B 0,C 180,E1 7514.012,E2 7514.012} C_VEL
LIN {X 0,Y 608.864,Z 780.81,A -85,B 0,C 180,E1 7519.825,E2 7519.825} C_VEL
LIN {X 0,Y 608.833,Z 780.81,A -85,B 0,C 180,E1 7525.2,E2 7525.2} C_VEL
LIN {X 0,Y 609.009,Z 780.81,A -85,B 0,C 180,E1 7530.276,E2 7530.276} C_VEL
LIN {X 0,Y 609.128,Z 780.81,A -85,B 0,C 180,E1 7535.063,E2 7535.063} C_VEL
LIN {X 0,Y 609.195,Z 780.81,A -85,B 0,C 180,E1 7540.488,E2 7540.488} C_VEL
LIN {X 0,Y 609.261,Z 780.81,A -85,B 0,C 180,E1 7545.644,E2 7545.644} C_VEL
LIN {X 0,Y 609.5,Z 780.81,A -85,B 0,C 180,E1 7551.449,E2 7551.449} C_VEL
LIN {X 0,Y 609.702,Z 780.81,A -85,B 0,C 180,E1 7557.161,E2 7557.161} C_VEL
LIN {X 0,Y 609.786,Z 780.81,A -85,B 0,C 180,E1 7561.422,E2 7561.422} C_VEL
LIN {X 0,Y 609.479,Z 780.81,A -85,B 0,C 180,E1 7567.122,E2 7567.122} C_VEL
LIN {X 0,Y 609.366,Z 780.81,A -85,B 0,C 180,E1 7571.443,E2 7571.443} C_VEL
LIN {X 0,Y 609.289,Z 780.81,A -85,B 0,C 180,E1 7577.314,E2 7577.314} C_VEL
LIN {X 0,Y 609.124,Z 780.81,A -85,B 0,C 180,E1 7581.845,E2 7581.845} C_VEL
LIN {X 0,Y 609.025,Z 780.81,A -85,B 0,C 180,E1 7586.72,E2 7586.72} C_VEL
LIN {X 0,Y 608.982,Z 780.81,A -85,B 0,C 180,E1 7592.473,E2 7592.473} C_VEL
LIN {X 0,Y 608.845,Z 780.81,A -85,B 0,C 180,E1 7598.346,E2 7598.346} C_VEL
LIN {X 0,Y 608.887,Z 780.81,A -85,B 0,C 180,E1 7604.012,E2 7604.012} C_VEL
LIN {X 0,Y 608.965,Z 781.397,A -85,B 0,C 180,E1 7609.284,E2 7609.284} C_VEL
LIN {X 0,Y 631.062,Z 827.97,A -85,B 0,C 180,E1 7611.691,E2 7611.691} C_VEL
LIN {X 0,Y 632.339,Z 833.101,A -85,B 0,C 180,E1 7611.912,E2 7611.912} C_VEL
LIN {X 0,Y 629.899,Z 875.567,A -85,B 0,C 180,E1 7613.15,E2 7613.15} C_VEL
LIN {X 0,Y 626.538,Z 916.939,A -85,B 0,C 180,E1 7614.927,E2 7614.927} C_VEL
LIN {X 0,Y 622.835,Z 956.179,A -85,B 0,C 180,E1 7617.221,E2 7617.221} C_VEL
LIN {X 0,Y 619.076,Z 992.83,A -85,B 0,C 180,E1 7620.029,E2 7620.029} C_VEL
LIN {X 0,Y 615.651,Z 1026.509,A -85,B 0,C 180,E1 7623.364,E2 7623.364} C_VEL
LIN {X 0,Y 613.013,Z 1056.373,A -85,B 0,C 180,E1 7627.158,E2 7627.158} C_VEL
LIN {X 0,Y 611.173,Z 1080.775,A -85,B 0,C 180,E1 7631.252,E2 7631.252} C_VEL
LIN {X 0,Y 610.335,Z 1096.954,A -85,B 0,C 180,E1 7634.897,E2 7634.897} C_VEL
LIN {X 0,Y 609.943,Z 1108.66,A -85,B 0,C 180,E1 7638.569,E2 7638.569} C_VEL
LIN {X 0,Y 609.692,Z 1116.333,A -85,B 0,C 180,E1 7642.418,E2 7642.418} C_VEL
LIN {X 0,Y 609.652,Z 1119.216,A -85,B 0,C 180,E1 7645.736,E2 7645.736} C_VEL
LIN {X 0,Y 609.757,Z 1118.07,A -85,B 0,C 180,E1 7650.001,E2 7650.001} C_VEL
LIN {X 0,Y 609.917,Z 1111.257,A -85,B 0,C 180,E1 7654.263,E2 7654.263} C_VEL
LIN {X 0,Y 610.237,Z 1100.133,A -85,B 0,C 180,E1 7658.153,E2 7658.153} C_VEL
LIN {X 0,Y 611.084,Z 1082.929,A -85,B 0,C 180,E1 7662.229,E2 7662.229} C_VEL
LIN {X 0,Y 612.528,Z 1060.83,A -85,B 0,C 180,E1 7666.077,E2 7666.077} C_VEL
LIN {X 0,Y 614.871,Z 1034.98,A -85,B 0,C 180,E1 7669.564,E2 7669.564} C_VEL
LIN {X 0,Y 618.138,Z 1002.336,A -85,B 0,C 180,E1 7673.026,E2 7673.026} C_VEL
LIN {X 0,Y 622,Z 964.672,A -85,B 0,C 180,E1 7676.106,E2 7676.106} C_VEL
LIN {X 0,Y 625.887,Z 924.513,A -85,B 0,C 180,E1 7678.587,E2 7678.587} C_VEL
LIN {X 0,Y 629.067,Z 885.633,A -85,B 0,C 180,E1 7680.378,E2 7680.378} C_VEL
LIN {X 0,Y 631.828,Z 843.596,A -85,B 0,C 180,E1 7681.747,E2 7681.747} C_VEL
LIN {X 0,Y 631.939,Z 829.974,A -85,B 0,C 180,E1 7682.106,E2 7682.106} C_VEL
LIN {X 0,Y 613.313,Z 790.711,A -85,B 0,C 180,E1 7684.118,E2 7684.118} C_VEL
LIN {X 0,Y 608.913,Z 780.81,A -85,B 0,C 180,E1 7684.604,E2 7684.604} C_VEL
LIN {X 0,Y 608.818,Z 780.81,A -85,B 0,C 180,E1 7690.191,E2 7690.191} C_VEL
LIN {X 0,Y 608.85,Z 780.81,A -85,B 0,C 180,E1 7696.035,E2 7696.035} C_VEL
LIN {X 0,Y 608.856,Z 780.81,A -85,B 0,C 180,E1 7701.655,E2 7701.655} C_VEL
LIN {X 0,Y 608.89,Z 780.81,A -85,B 0,C 180,E1 7707.544,E2 7707.544} C_VEL
LIN {X 0,Y 609.079,Z 780.81,A -85,B 0,C 180,E1 7713.273,E2 7713.273} C_VEL
LIN {X 0,Y 609.144,Z 780.81,A -85,B 0,C 180,E1 7718.156,E2 7718.156} C_VEL
LIN {X 0,Y 609.29,Z 780.81,A -85,B 0,C 180,E1 7722.687,E2 7722.687} C_VEL
LIN {X 0,Y 609.366,Z 780.81,A -85,B 0,C 180,E1 7728.557,E2 7728.557} C_VEL
LIN {X 0,Y 609.517,Z 780.81,A -85,B 0,C 180,E1 7733.12,E2 7733.12} C_VEL
LIN {X 0,Y 609.663,Z 780.81,A -85,B 0,C 180,E1 7738.578,E2 7738.578} C_VEL
LIN {X 0,Y 609.563,Z 780.81,A -85,B 0,C 180,E1 7742.839,E2 7742.839} C_VEL
LIN {X 0,Y 609.503,Z 780.81,A -85,B 0,C 180,E1 7748.551,E2 7748.551} C_VEL
LIN {X 0,Y 609.325,Z 780.81,A -85,B 0,C 180,E1 7754.354,E2 7754.354} C_VEL
LIN {X 0,Y 609.246,Z 780.81,A -85,B 0,C 180,E1 7759.521,E2 7759.521} C_VEL
LIN {X 0,Y 609.118,Z 780.81,A -85,B 0,C 180,E1 7764.937,E2 7764.937} C_VEL
LIN {X 0,Y 609.052,Z 780.81,A -85,B 0,C 180,E1 7769.742,E2 7769.742} C_VEL
LIN {X 0,Y 608.935,Z 780.81,A -85,B 0,C 180,E1 7775.023,E2 7775.023} C_VEL
LIN {X 0,Y 608.784,Z 780.81,A -85,B 0,C 180,E1 7780.182,E2 7780.182} C_VEL
LIN {X 0,Y 608.807,Z 780.81,A -85,B 0,C 180,E1 7786.025,E2 7786.025} C_VEL
LIN {X 0,Y 608.797,Z 780.81,A -85,B 0,C 180,E1 7790.239,E2 7790.239} C_VEL
LIN {X 0,Y 608.684,Z 783.549,A -85,B 0,C 180,E1 7790.983,E2 7790.983} C_VEL
LIN {X 0,Y 609.052,Z 793.295,A -85,B 0,C 180,E1 7791.836,E2 7791.836} C_VEL
LIN {X 0,Y 612.654,Z 804.629,A -85,B 0,C 180,E1 7792.492,E2 7792.492} C_VEL
LIN {X 0,Y 627,Z 835.085,A -85,B 0,C 180,E1 7793.896,E2 7793.896} C_VEL
LIN {X 0,Y 624.964,Z 880.443,A -85,B 0,C 180,E1 7794.774,E2 7794.774} C_VEL
LIN {X 0,Y 621.923,Z 925.09,A -85,B 0,C 180,E1 7796.242,E2 7796.242} C_VEL
LIN {X 0,Y 618.213,Z 966.579,A -85,B 0,C 180,E1 7798.193,E2 7798.193} C_VEL
LIN {X 0,Y 614.436,Z 1005.151,A -85,B 0,C 180,E1 7800.62,E2 7800.62} C_VEL
LIN {X 0,Y 610.571,Z 1042.635,A -85,B 0,C 180,E1 7803.687,E2 7803.687} C_VEL
LIN {X 0,Y 607.049,Z 1076.796,A -85,B 0,C 180,E1 7807.312,E2 7807.312} C_VEL
LIN {X 0,Y 604.613,Z 1104.921,A -85,B 0,C 180,E1 7811.263,E2 7811.263} C_VEL
LIN {X 0,Y 603.01,Z 1127.456,A -85,B 0,C 180,E1 7815.487,E2 7815.487} C_VEL
LIN {X 0,Y 602.188,Z 1142.956,A -85,B 0,C 180,E1 7819.517,E2 7819.517} C_VEL
LIN {X 0,Y 601.962,Z 1153.235,A -85,B 0,C 180,E1 7823.513,E2 7823.513} C_VEL
LIN {X 0,Y 601.895,Z 1158.218,A -85,B 0,C 180,E1 7827.121,E2 7827.121} C_VEL
LIN {X 0,Y 601.898,Z 1159.167,A -85,B 0,C 180,E1 7831.438,E2 7831.438} C_VEL
LIN {X 0,Y 601.956,Z 1154.487,A -85,B 0,C 180,E1 7835.762,E2 7835.762} C_VEL
LIN {X 0,Y 602.144,Z 1145.252,A -85,B 0,C 180,E1 7839.752,E2 7839.752} C_VEL
LIN {X 0,Y 602.803,Z 1130.699,A -85,B 0,C 180,E1 7843.776,E2 7843.776} C_VEL
LIN {X 0,Y 604.036,Z 1111.301,A -85,B 0,C 180,E1 7847.658,E2 7847.658} C_VEL
LIN {X 0,Y 606.368,Z 1085.69,A -85,B 0,C 180,E1 7851.545,E2 7851.545} C_VEL
LIN {X 0,Y 609.449,Z 1053.523,A -85,B 0,C 180,E1 7855.256,E2 7855.256} C_VEL
LIN {X 0,Y 613.3,Z 1016.464,A -85,B 0,C 180,E1 7858.539,E2 7858.539} C_VEL
LIN {X 0,Y 617.338,Z 976.156,A -85,B 0,C 180,E1 7861.264,E2 7861.264} C_VEL
LIN {X 0,Y 621.04,Z 935.696,A -85,B 0,C 180,E1 7863.311,E2 7863.311} C_VEL
LIN {X 0,Y 624.153,Z 894.623,A -85,B 0,C 180,E1 7864.82,E2 7864.82} C_VEL
LIN {X 0,Y 626.536,Z 849.614,A -85,B 0,C 180,E1 7865.882,E2 7865.882} C_VEL
LIN {X 0,Y 626.385,Z 832.535,A -85,B 0,C 180,E1 7866.189,E2 7866.189} C_VEL
LIN {X 0,Y 602.982,Z 786.086,A -85,B 0,C 180,E1 7868.563,E2 7868.563} C_VEL
LIN {X 0,Y 600.932,Z 780.81,A -85,B 0,C 180,E1 7868.849,E2 7868.849} C_VEL
LIN {X 0,Y 600.944,Z 780.81,A -85,B 0,C 180,E1 7874.754,E2 7874.754} C_VEL
LIN {X 0,Y 600.906,Z 780.81,A -85,B 0,C 180,E1 7879.181,E2 7879.181} C_VEL
LIN {X 0,Y 600.923,Z 780.81,A -85,B 0,C 180,E1 7884.674,E2 7884.674} C_VEL
LIN {X 0,Y 601.035,Z 780.81,A -85,B 0,C 180,E1 7889.821,E2 7889.821} C_VEL
LIN {X 0,Y 601.22,Z 780.81,A -85,B 0,C 180,E1 7894.797,E2 7894.797} C_VEL
LIN {X 0,Y 601.241,Z 780.81,A -85,B 0,C 180,E1 7899.405,E2 7899.405} C_VEL
LIN {X 0,Y 601.376,Z 780.81,A -85,B 0,C 180,E1 7903.96,E2 7903.96} C_VEL
LIN {X 0,Y 601.46,Z 780.81,A -85,B 0,C 180,E1 7909.875,E2 7909.875} C_VEL
LIN {X 0,Y 601.577,Z 780.81,A -85,B 0,C 180,E1 7914.237,E2 7914.237} C_VEL
LIN {X 0,Y 601.709,Z 780.81,A -85,B 0,C 180,E1 7918.563,E2 7918.563} C_VEL
LIN {X 0,Y 601.664,Z 780.81,A -85,B 0,C 180,E1 7922.881,E2 7922.881} C_VEL
LIN {X 0,Y 601.595,Z 780.81,A -85,B 0,C 180,E1 7927.216,E2 7927.216} C_VEL
LIN {X 0,Y 601.448,Z 780.81,A -85,B 0,C 180,E1 7933.069,E2 7933.069} C_VEL
LIN {X 0,Y 601.365,Z 780.81,A -85,B 0,C 180,E1 7937.549,E2 7937.549} C_VEL
LIN {X 0,Y 601.19,Z 780.81,A -85,B 0,C 180,E1 7942.148,E2 7942.148} C_VEL
LIN {X 0,Y 601.105,Z 780.81,A -85,B 0,C 180,E1 7946.902,E2 7946.902} C_VEL
LIN {X 0,Y 601.054,Z 780.81,A -85,B 0,C 180,E1 7951.864,E2 7951.864} C_VEL
LIN {X 0,Y 600.92,Z 780.81,A -85,B 0,C 180,E1 7957.117,E2 7957.117} C_VEL
LIN {X 0,Y 600.91,Z 780.81,A -85,B 0,C 180,E1 7963.177,E2 7963.177} C_VEL
LIN {X 0,Y 601,Z 780.81,A -85,B 0,C 180,E1 7968.652,E2 7968.652} C_VEL
LIN {X 0,Y 605.532,Z 790.777,A -85,B 0,C 180,E1 7969.163,E2 7969.163} C_VEL
LIN {X 0,Y 623.943,Z 829.205,A -85,B 0,C 180,E1 7971.25,E2 7971.25} C_VEL
LIN {X 0,Y 625.789,Z 835.827,A -85,B 0,C 180,E1 7971.555,E2 7971.555} C_VEL
LIN {X 0,Y 623.212,Z 877.2,A -85,B 0,C 180,E1 7972.795,E2 7972.795} C_VEL
LIN {X 0,Y 619.631,Z 919.184,A -85,B 0,C 180,E1 7974.635,E2 7974.635} C_VEL
LIN {X 0,Y 615.687,Z 958.182,A -85,B 0,C 180,E1 7976.967,E2 7976.967} C_VEL
LIN {X 0,Y 611.891,Z 993.121,A -85,B 0,C 180,E1 7979.687,E2 7979.687} C_VEL
LIN {X 0,Y 608.264,Z 1026.579,A -85,B 0,C 180,E1 7983.04,E2 7983.04} C_VEL
LIN {X 0,Y 605.276,Z 1057.42,A -85,B 0,C 180,E1 7987.056,E2 7987.056} C_VEL
LIN {X 0,Y 603.41,Z 1080.549,A -85,B 0,C 180,E1 7991.002,E2 7991.002} C_VEL
LIN {X 0,Y 602.479,Z 1096.801,A -85,B 0,C 180,E1 7994.695,E2 7994.695} C_VEL
LIN {X 0,Y 602.052,Z 1108.551,A -85,B 0,C 180,E1 7998.417,E2 7998.417} C_VEL
LIN {X 0,Y 601.794,Z 1116.285,A -85,B 0,C 180,E1 8002.318,E2 8002.318} C_VEL
LIN {X 0,Y 601.749,Z 1119.206,A -85,B 0,C 180,E1 8005.68,E2 8005.68} C_VEL
LIN {X 0,Y 601.872,Z 1118.098,A -85,B 0,C 180,E1 8010.001,E2 8010.001} C_VEL
LIN {X 0,Y 602.019,Z 1112.898,A -85,B 0,C 180,E1 8013.599,E2 8013.599} C_VEL
LIN {X 0,Y 602.348,Z 1101,A -85,B 0,C 180,E1 8018.057,E2 8018.057} C_VEL
LIN {X 0,Y 603.285,Z 1083.158,A -85,B 0,C 180,E1 8022.382,E2 8022.382} C_VEL
LIN {X 0,Y 604.899,Z 1060.859,A -85,B 0,C 180,E1 8026.323,E2 8026.323} C_VEL
LIN {X 0,Y 607.476,Z 1033.885,A -85,B 0,C 180,E1 8030.002,E2 8030.002} C_VEL
LIN {X 0,Y 610.89,Z 1001.996,A -85,B 0,C 180,E1 8033.419,E2 8033.419} C_VEL
LIN {X 0,Y 615.093,Z 964.01,A -85,B 0,C 180,E1 8036.54,E2 8036.54} C_VEL
LIN {X 0,Y 619.4,Z 921.933,A -85,B 0,C 180,E1 8039.131,E2 8039.131} C_VEL
LIN {X 0,Y 622.907,Z 880.631,A -85,B 0,C 180,E1 8040.981,E2 8040.981} C_VEL
LIN {X 0,Y 625.589,Z 839.763,A -85,B 0,C 180,E1 8042.258,E2 8042.258} C_VEL
LIN {X 0,Y 624.984,Z 831.755,A -85,B 0,C 180,E1 8042.515,E2 8042.515} C_VEL
LIN {X 0,Y 605.931,Z 791.575,A -85,B 0,C 180,E1 8044.627,E2 8044.627} C_VEL
LIN {X 0,Y 600.965,Z 780.81,A -85,B 0,C 180,E1 8045.221,E2 8045.221} C_VEL
LIN {X 0,Y 600.89,Z 780.81,A -85,B 0,C 180,E1 8051.032,E2 8051.032} C_VEL
LIN {X 0,Y 600.868,Z 780.81,A -85,B 0,C 180,E1 8056.83,E2 8056.83} C_VEL
LIN {X 0,Y 600.901,Z 780.81,A -85,B 0,C 180,E1 8062.881,E2 8062.881} C_VEL
LIN {X 0,Y 600.999,Z 780.81,A -85,B 0,C 180,E1 8068.747,E2 8068.747} C_VEL
LIN {X 0,Y 601.179,Z 780.81,A -85,B 0,C 180,E1 8073.102,E2 8073.102} C_VEL
LIN {X 0,Y 601.228,Z 780.81,A -85,B 0,C 180,E1 8078.428,E2 8078.428} C_VEL
LIN {X 0,Y 601.374,Z 780.81,A -85,B 0,C 180,E1 8083.955,E2 8083.955} C_VEL
LIN {X 0,Y 601.493,Z 780.81,A -85,B 0,C 180,E1 8089.871,E2 8089.871} C_VEL
LIN {X 0,Y 601.606,Z 780.81,A -85,B 0,C 180,E1 8094.232,E2 8094.232} C_VEL
LIN {X 0,Y 601.765,Z 780.81,A -85,B 0,C 180,E1 8098.559,E2 8098.559} C_VEL
LIN {X 0,Y 601.66,Z 780.81,A -85,B 0,C 180,E1 8102.877,E2 8102.877} C_VEL
LIN {X 0,Y 601.583,Z 780.81,A -85,B 0,C 180,E1 8108.665,E2 8108.665} C_VEL
LIN {X 0,Y 601.433,Z 780.81,A -85,B 0,C 180,E1 8114.547,E2 8114.547} C_VEL
LIN {X 0,Y 601.343,Z 780.81,A -85,B 0,C 180,E1 8119.061,E2 8119.061} C_VEL
LIN {X 0,Y 601.189,Z 780.81,A -85,B 0,C 180,E1 8123.707,E2 8123.707} C_VEL
LIN {X 0,Y 601.146,Z 780.81,A -85,B 0,C 180,E1 8128.521,E2 8128.521} C_VEL
LIN {X 0,Y 601.025,Z 780.81,A -85,B 0,C 180,E1 8133.932,E2 8133.932} C_VEL
LIN {X 0,Y 600.913,Z 780.81,A -85,B 0,C 180,E1 8138.941,E2 8138.941} C_VEL
LIN {X 0,Y 600.802,Z 780.81,A -85,B 0,C 180,E1 8144.755,E2 8144.755} C_VEL
LIN {X 0,Y 600.797,Z 780.81,A -85,B 0,C 180,E1 8150.243,E2 8150.243} C_VEL
LIN {X 0,Y 600.925,Z 780.81,A -85,B 0,C 180,E1 8151.289,E2 8151.289} C_VEL
LIN {X 0,Y 607.711,Z 795.313,A -85,B 0,C 180,E1 8152.012,E2 8152.012} C_VEL
LIN {X 0,Y 612.654,Z 804.629,A -85,B 0,C 180,E1 8152.492,E2 8152.492} C_VEL
LIN {X 0,Y 614.704,Z 812.679,A -85,B 0,C 180,E1 8152.748,E2 8152.748} C_VEL
LIN {X 0,Y 616.233,Z 827.256,A -85,B 0,C 180,E1 8153.058,E2 8153.058} C_VEL
LIN {X 0,Y 620.521,Z 836.537,A -85,B 0,C 180,E1 8153.493,E2 8153.493} C_VEL
LIN {X 0,Y 618.393,Z 880.883,A -85,B 0,C 180,E1 8154.37,E2 8154.37} C_VEL
LIN {X 0,Y 615.309,Z 924.523,A -85,B 0,C 180,E1 8155.817,E2 8155.817} C_VEL
LIN {X 0,Y 611.49,Z 964.564,A -85,B 0,C 180,E1 8157.696,E2 8157.696} C_VEL
LIN {X 0,Y 607.471,Z 1003.803,A -85,B 0,C 180,E1 8160.164,E2 8160.164} C_VEL
LIN {X 0,Y 603.281,Z 1041.926,A -85,B 0,C 180,E1 8163.3,E2 8163.3} C_VEL
LIN {X 0,Y 599.488,Z 1076.787,A -85,B 0,C 180,E1 8167.046,E2 8167.046} C_VEL
LIN {X 0,Y 597.023,Z 1104.705,A -85,B 0,C 180,E1 8170.982,E2 8170.982} C_VEL
LIN {X 0,Y 595.305,Z 1125.853,A -85,B 0,C 180,E1 8174.947,E2 8174.947} C_VEL
LIN {X 0,Y 594.366,Z 1141.81,A -85,B 0,C 180,E1 8179.007,E2 8179.007} C_VEL
LIN {X 0,Y 594.07,Z 1153.235,A -85,B 0,C 180,E1 8183.426,E2 8183.426} C_VEL
LIN {X 0,Y 593.988,Z 1158.218,A -85,B 0,C 180,E1 8187.083,E2 8187.083} C_VEL
LIN {X 0,Y 593.994,Z 1159.166,A -85,B 0,C 180,E1 8191.457,E2 8191.457} C_VEL
LIN {X 0,Y 594.055,Z 1154.487,A -85,B 0,C 180,E1 8195.839,E2 8195.839} C_VEL
LIN {X 0,Y 594.269,Z 1145.252,A -85,B 0,C 180,E1 8199.882,E2 8199.882} C_VEL
LIN {X 0,Y 595.107,Z 1129.164,A -85,B 0,C 180,E1 8204.333,E2 8204.333} C_VEL
LIN {X 0,Y 596.694,Z 1108.025,A -85,B 0,C 180,E1 8208.46,E2 8208.46} C_VEL
LIN {X 0,Y 598.872,Z 1083.995,A -85,B 0,C 180,E1 8212.025,E2 8212.025} C_VEL
LIN {X 0,Y 602.088,Z 1053.322,A -85,B 0,C 180,E1 8215.577,E2 8215.577} C_VEL
LIN {X 0,Y 606.157,Z 1015.999,A -85,B 0,C 180,E1 8218.921,E2 8218.921} C_VEL
LIN {X 0,Y 610.373,Z 976.225,A -85,B 0,C 180,E1 8221.636,E2 8221.636} C_VEL
LIN {X 0,Y 614.302,Z 935.595,A -85,B 0,C 180,E1 8223.715,E2 8223.715} C_VEL
LIN {X 0,Y 617.643,Z 894.19,A -85,B 0,C 180,E1 8225.249,E2 8225.249} C_VEL
LIN {X 0,Y 620.191,Z 848.463,A -85,B 0,C 180,E1 8226.333,E2 8226.333} C_VEL
LIN {X 0,Y 619.827,Z 834.784,A -85,B 0,C 180,E1 8226.599,E2 8226.599} C_VEL
LIN {X 0,Y 597.462,Z 790.576,A -85,B 0,C 180,E1 8228.928,E2 8228.928} C_VEL
LIN {X 0,Y 592.969,Z 780.81,A -85,B 0,C 180,E1 8229.475,E2 8229.475} C_VEL
LIN {X 0,Y 593.039,Z 780.81,A -85,B 0,C 180,E1 8234.496,E2 8234.496} C_VEL
LIN {X 0,Y 592.962,Z 780.81,A -85,B 0,C 180,E1 8240.435,E2 8240.435} C_VEL
LIN {X 0,Y 593.005,Z 780.81,A -85,B 0,C 180,E1 8245.912,E2 8245.912} C_VEL
LIN {X 0,Y 593.16,Z 780.81,A -85,B 0,C 180,E1 8251.059,E2 8251.059} C_VEL
LIN {X 0,Y 593.283,Z 780.81,A -85,B 0,C 180,E1 8256.479,E2 8256.479} C_VEL
LIN {X 0,Y 593.414,Z 780.81,A -85,B 0,C 180,E1 8262.213,E2 8262.213} C_VEL
LIN {X 0,Y 593.427,Z 780.81,A -85,B 0,C 180,E1 8266.756,E2 8266.756} C_VEL
LIN {X 0,Y 593.712,Z 780.81,A -85,B 0,C 180,E1 8272.692,E2 8272.692} C_VEL
LIN {X 0,Y 593.809,Z 780.81,A -85,B 0,C 180,E1 8278.544,E2 8278.544} C_VEL
LIN {X 0,Y 593.761,Z 780.81,A -85,B 0,C 180,E1 8282.919,E2 8282.919} C_VEL
LIN {X 0,Y 593.708,Z 780.81,A -85,B 0,C 180,E1 8288.785,E2 8288.785} C_VEL
LIN {X 0,Y 593.539,Z 780.81,A -85,B 0,C 180,E1 8294.749,E2 8294.749} C_VEL
LIN {X 0,Y 593.348,Z 780.81,A -85,B 0,C 180,E1 8299.562,E2 8299.562} C_VEL
LIN {X 0,Y 593.224,Z 780.81,A -85,B 0,C 180,E1 8304.05,E2 8304.05} C_VEL
LIN {X 0,Y 593.132,Z 780.81,A -85,B 0,C 180,E1 8308.948,E2 8308.948} C_VEL
LIN {X 0,Y 593.06,Z 780.81,A -85,B 0,C 180,E1 8314.09,E2 8314.09} C_VEL
LIN {X 0,Y 592.936,Z 780.81,A -85,B 0,C 180,E1 8320.134,E2 8320.134} C_VEL
LIN {X 0,Y 592.976,Z 780.81,A -85,B 0,C 180,E1 8325.516,E2 8325.516} C_VEL
LIN {X 0,Y 593.136,Z 780.81,A -85,B 0,C 180,E1 8328.012,E2 8328.012} C_VEL
LIN {X 0,Y 597.71,Z 790.875,A -85,B 0,C 180,E1 8328.556,E2 8328.556} C_VEL
LIN {X 0,Y 616.35,Z 829.065,A -85,B 0,C 180,E1 8330.719,E2 8330.719} C_VEL
LIN {X 0,Y 619.288,Z 837.678,A -85,B 0,C 180,E1 8331.164,E2 8331.164} C_VEL
LIN {X 0,Y 616.65,Z 877.62,A -85,B 0,C 180,E1 8332.385,E2 8332.385} C_VEL
LIN {X 0,Y 612.865,Z 919.596,A -85,B 0,C 180,E1 8334.241,E2 8334.241} C_VEL
LIN {X 0,Y 608.72,Z 958.791,A -85,B 0,C 180,E1 8336.613,E2 8336.613} C_VEL
LIN {X 0,Y 604.603,Z 994.494,A -85,B 0,C 180,E1 8339.436,E2 8339.436} C_VEL
LIN {X 0,Y 600.973,Z 1026.505,A -85,B 0,C 180,E1 8342.686,E2 8342.686} C_VEL
LIN {X 0,Y 597.735,Z 1056.846,A -85,B 0,C 180,E1 8346.693,E2 8346.693} C_VEL
LIN {X 0,Y 595.664,Z 1080.323,A -85,B 0,C 180,E1 8350.745,E2 8350.745} C_VEL
LIN {X 0,Y 594.675,Z 1096.369,A -85,B 0,C 180,E1 8354.411,E2 8354.411} C_VEL
LIN {X 0,Y 594.178,Z 1108.443,A -85,B 0,C 180,E1 8358.262,E2 8358.262} C_VEL
LIN {X 0,Y 593.921,Z 1115.873,A -85,B 0,C 180,E1 8361.957,E2 8361.957} C_VEL
LIN {X 0,Y 593.841,Z 1119.196,A -85,B 0,C 180,E1 8365.623,E2 8365.623} C_VEL
LIN {X 0,Y 593.971,Z 1118.126,A -85,B 0,C 180,E1 8370.001,E2 8370.001} C_VEL
LIN {X 0,Y 594.119,Z 1112.985,A -85,B 0,C 180,E1 8373.646,E2 8373.646} C_VEL
LIN {X 0,Y 594.488,Z 1101.436,A -85,B 0,C 180,E1 8378.065,E2 8378.065} C_VEL
LIN {X 0,Y 595.356,Z 1085.274,A -85,B 0,C 180,E1 8382.133,E2 8382.133} C_VEL
LIN {X 0,Y 596.845,Z 1065.495,A -85,B 0,C 180,E1 8385.853,E2 8385.853} C_VEL
LIN {X 0,Y 599.684,Z 1037.561,A -85,B 0,C 180,E1 8389.889,E2 8389.889} C_VEL
LIN {X 0,Y 603.321,Z 1005.622,A -85,B 0,C 180,E1 8393.43,E2 8393.43} C_VEL
LIN {X 0,Y 607.312,Z 970.975,A -85,B 0,C 180,E1 8396.41,E2 8396.41} C_VEL
LIN {X 0,Y 611.473,Z 933.346,A -85,B 0,C 180,E1 8398.909,E2 8398.909} C_VEL
LIN {X 0,Y 615.39,Z 892.182,A -85,B 0,C 180,E1 8400.953,E2 8400.953} C_VEL
LIN {X 0,Y 618.621,Z 848.24,A -85,B 0,C 180,E1 8402.463,E2 8402.463} C_VEL
LIN {X 0,Y 618.668,Z 835.06,A -85,B 0,C 180,E1 8402.846,E2 8402.846} C_VEL
LIN {X 0,Y 599.859,Z 795.19,A -85,B 0,C 180,E1 8405.013,E2 8405.013} C_VEL
LIN {X 0,Y 593.095,Z 781.864,A -85,B 0,C 180,E1 8405.715,E2 8405.715} C_VEL
LIN {X 0,Y 593.026,Z 780.81,A -85,B 0,C 180,E1 8405.88,E2 8405.88} C_VEL
LIN {X 0,Y 592.958,Z 780.81,A -85,B 0,C 180,E1 8411.499,E2 8411.499} C_VEL
LIN {X 0,Y 592.936,Z 780.81,A -85,B 0,C 180,E1 8416.527,E2 8416.527} C_VEL
LIN {X 0,Y 592.949,Z 780.81,A -85,B 0,C 180,E1 8422.297,E2 8422.297} C_VEL
LIN {X 0,Y 593.004,Z 780.81,A -85,B 0,C 180,E1 8427.651,E2 8427.651} C_VEL
LIN {X 0,Y 593.28,Z 780.81,A -85,B 0,C 180,E1 8433.059,E2 8433.059} C_VEL
LIN {X 0,Y 593.34,Z 780.81,A -85,B 0,C 180,E1 8439.113,E2 8439.113} C_VEL
LIN {X 0,Y 593.463,Z 780.81,A -85,B 0,C 180,E1 8443.735,E2 8443.735} C_VEL
LIN {X 0,Y 593.593,Z 780.81,A -85,B 0,C 180,E1 8449.735,E2 8449.735} C_VEL
LIN {X 0,Y 593.7,Z 780.81,A -85,B 0,C 180,E1 8454.155,E2 8454.155} C_VEL
LIN {X 0,Y 593.864,Z 780.81,A -85,B 0,C 180,E1 8458.54,E2 8458.54} C_VEL
LIN {X 0,Y 593.757,Z 780.81,A -85,B 0,C 180,E1 8462.915,E2 8462.915} C_VEL
LIN {X 0,Y 593.687,Z 780.81,A -85,B 0,C 180,E1 8468.781,E2 8468.781} C_VEL
LIN {X 0,Y 593.509,Z 780.81,A -85,B 0,C 180,E1 8474.745,E2 8474.745} C_VEL
LIN {X 0,Y 593.386,Z 780.81,A -85,B 0,C 180,E1 8479.567,E2 8479.567} C_VEL
LIN {X 0,Y 593.252,Z 780.81,A -85,B 0,C 180,E1 8484.044,E2 8484.044} C_VEL
LIN {X 0,Y 593.187,Z 780.81,A -85,B 0,C 180,E1 8488.94,E2 8488.94} C_VEL
LIN {X 0,Y 593.114,Z 780.81,A -85,B 0,C 180,E1 8494.081,E2 8494.081} C_VEL
LIN {X 0,Y 592.898,Z 780.81,A -85,B 0,C 180,E1 8500.127,E2 8500.127} C_VEL
LIN {X 0,Y 592.91,Z 780.81,A -85,B 0,C 180,E1 8505.517,E2 8505.517} C_VEL
LIN {X 0,Y 592.954,Z 780.872,A -85,B 0,C 180,E1 8510.718,E2 8510.718} C_VEL
LIN {X 0,Y 597.491,Z 790.817,A -85,B 0,C 180,E1 8511.206,E2 8511.206} C_VEL
LIN {X 0,Y 616.233,Z 827.256,A -85,B 0,C 180,E1 8513.058,E2 8513.058} C_VEL
LIN {X 0,Y 617.411,Z 838.094,A -85,B 0,C 180,E1 8513.304,E2 8513.304} C_VEL
LIN {X 0,Y 612.961,Z 862.281,A -85,B 0,C 180,E1 8513.505,E2 8513.505} C_VEL
LIN {X 0,Y 609.772,Z 909.125,A -85,B 0,C 180,E1 8514.815,E2 8514.815} C_VEL
LIN {X 0,Y 605.934,Z 952.439,A -85,B 0,C 180,E1 8516.667,E2 8516.667} C_VEL
LIN {X 0,Y 601.903,Z 990.729,A -85,B 0,C 180,E1 8518.893,E2 8518.893} C_VEL
LIN {X 0,Y 597.517,Z 1028.766,A -85,B 0,C 180,E1 8521.78,E2 8521.78} C_VEL
LIN {X 0,Y 593.349,Z 1065.02,A -85,B 0,C 180,E1 8525.377,E2 8525.377} C_VEL
LIN {X 0,Y 590.006,Z 1096.201,A -85,B 0,C 180,E1 8529.42,E2 8529.42} C_VEL
LIN {X 0,Y 587.962,Z 1120.35,A -85,B 0,C 180,E1 8533.577,E2 8533.577} C_VEL
LIN {X 0,Y 586.758,Z 1137.952,A -85,B 0,C 180,E1 8537.732,E2 8537.732} C_VEL
LIN {X 0,Y 586.251,Z 1150.115,A -85,B 0,C 180,E1 8541.849,E2 8541.849} C_VEL
LIN {X 0,Y 586.042,Z 1156.659,A -85,B 0,C 180,E1 8545.563,E2 8545.563} C_VEL
LIN {X 0,Y 586.049,Z 1159.5,A -85,B 0,C 180,E1 8549.999,E2 8549.999} C_VEL
LIN {X 0,Y 586.027,Z 1156.662,A -85,B 0,C 180,E1 8554.436,E2 8554.436} C_VEL
LIN {X 0,Y 586.268,Z 1150.119,A -85,B 0,C 180,E1 8558.149,E2 8558.149} C_VEL
LIN {X 0,Y 586.842,Z 1136.893,A -85,B 0,C 180,E1 8562.566,E2 8562.566} C_VEL
LIN {X 0,Y 587.952,Z 1120.354,A -85,B 0,C 180,E1 8566.421,E2 8566.421} C_VEL
LIN {X 0,Y 589.979,Z 1096.231,A -85,B 0,C 180,E1 8570.574,E2 8570.574} C_VEL
LIN {X 0,Y 593.325,Z 1065.006,A -85,B 0,C 180,E1 8574.623,E2 8574.623} C_VEL
LIN {X 0,Y 597.498,Z 1028.689,A -85,B 0,C 180,E1 8578.224,E2 8578.224} C_VEL
LIN {X 0,Y 602.06,Z 989.024,A -85,B 0,C 180,E1 8581.221,E2 8581.221} C_VEL
LIN {X 0,Y 606.471,Z 947.559,A -85,B 0,C 180,E1 8583.572,E2 8583.572} C_VEL
LIN {X 0,Y 610.149,Z 906.04,A -85,B 0,C 180,E1 8585.293,E2 8585.293} C_VEL
LIN {X 0,Y 613.184,Z 861.412,A -85,B 0,C 180,E1 8586.529,E2 8586.529} C_VEL
LIN {X 0,Y 613.666,Z 837.879,A -85,B 0,C 180,E1 8586.98,E2 8586.98} C_VEL
LIN {X 0,Y 590.342,Z 791.687,A -85,B 0,C 180,E1 8589.486,E2 8589.486} C_VEL
LIN {X 0,Y 585.114,Z 781.647,A -85,B 0,C 180,E1 8590.08,E2 8590.08} C_VEL
LIN {X 0,Y 585.067,Z 780.81,A -85,B 0,C 180,E1 8590.217,E2 8590.217} C_VEL
LIN {X 0,Y 585.119,Z 780.81,A -85,B 0,C 180,E1 8595.803,E2 8595.803} C_VEL
LIN {X 0,Y 585.029,Z 780.81,A -85,B 0,C 180,E1 8601.701,E2 8601.701} C_VEL
LIN {X 0,Y 585.091,Z 780.81,A -85,B 0,C 180,E1 8607.164,E2 8607.164} C_VEL
LIN {X 0,Y 585.274,Z 780.81,A -85,B 0,C 180,E1 8612.314,E2 8612.314} C_VEL
LIN {X 0,Y 585.351,Z 780.81,A -85,B 0,C 180,E1 8617.224,E2 8617.224} C_VEL
LIN {X 0,Y 585.511,Z 780.81,A -85,B 0,C 180,E1 8622.725,E2 8622.725} C_VEL
LIN {X 0,Y 585.601,Z 780.81,A -85,B 0,C 180,E1 8628.681,E2 8628.681} C_VEL
LIN {X 0,Y 585.795,Z 780.81,A -85,B 0,C 180,E1 8634.081,E2 8634.081} C_VEL
LIN {X 0,Y 585.908,Z 780.81,A -85,B 0,C 180,E1 8638.525,E2 8638.525} C_VEL
LIN {X 0,Y 585.859,Z 780.81,A -85,B 0,C 180,E1 8642.959,E2 8642.959} C_VEL
LIN {X 0,Y 585.789,Z 780.81,A -85,B 0,C 180,E1 8647.412,E2 8647.412} C_VEL
LIN {X 0,Y 585.631,Z 780.81,A -85,B 0,C 180,E1 8651.913,E2 8651.913} C_VEL
LIN {X 0,Y 585.524,Z 780.81,A -85,B 0,C 180,E1 8657.279,E2 8657.279} C_VEL
LIN {X 0,Y 585.324,Z 780.81,A -85,B 0,C 180,E1 8662.782,E2 8662.782} C_VEL
LIN {X 0,Y 585.216,Z 780.81,A -85,B 0,C 180,E1 8668.609,E2 8668.609} C_VEL
LIN {X 0,Y 585.133,Z 780.81,A -85,B 0,C 180,E1 8674.617,E2 8674.617} C_VEL
LIN {X 0,Y 585.038,Z 780.81,A -85,B 0,C 180,E1 8680.215,E2 8680.215} C_VEL
LIN {X 0,Y 585.067,Z 780.81,A -85,B 0,C 180,E1 8685.786,E2 8685.786} C_VEL
LIN {X 0,Y 585.123,Z 780.81,A -85,B 0,C 180,E1 8687.337,E2 8687.337} C_VEL
LIN {X 0,Y 589.893,Z 790.968,A -85,B 0,C 180,E1 8687.926,E2 8687.926} C_VEL
LIN {X 0,Y 608.449,Z 828.314,A -85,B 0,C 180,E1 8690.126,E2 8690.126} C_VEL
LIN {X 0,Y 612.737,Z 841.117,A -85,B 0,C 180,E1 8690.8,E2 8690.8} C_VEL
LIN {X 0,Y 609.859,Z 881.385,A -85,B 0,C 180,E1 8692.094,E2 8692.094} C_VEL
LIN {X 0,Y 605.901,Z 922.762,A -85,B 0,C 180,E1 8693.982,E2 8693.982} C_VEL
LIN {X 0,Y 601.267,Z 963.993,A -85,B 0,C 180,E1 8696.57,E2 8696.57} C_VEL
LIN {X 0,Y 596.65,Z 1001.224,A -85,B 0,C 180,E1 8699.673,E2 8699.673} C_VEL
LIN {X 0,Y 592.661,Z 1033.401,A -85,B 0,C 180,E1 8703.161,E2 8703.161} C_VEL
LIN {X 0,Y 589.812,Z 1059.993,A -85,B 0,C 180,E1 8706.881,E2 8706.881} C_VEL
LIN {X 0,Y 587.779,Z 1082.051,A -85,B 0,C 180,E1 8710.866,E2 8710.866} C_VEL
LIN {X 0,Y 586.666,Z 1099.334,A -85,B 0,C 180,E1 8715.075,E2 8715.075} C_VEL
LIN {X 0,Y 586.259,Z 1110.446,A -85,B 0,C 180,E1 8718.964,E2 8718.964} C_VEL
LIN {X 0,Y 586.01,Z 1116.748,A -85,B 0,C 180,E1 8722.593,E2 8722.593} C_VEL
LIN {X 0,Y 586.021,Z 1119.487,A -85,B 0,C 180,E1 8727.045,E2 8727.045} C_VEL
LIN {X 0,Y 586.163,Z 1116.557,A -85,B 0,C 180,E1 8731.478,E2 8731.478} C_VEL
LIN {X 0,Y 586.249,Z 1109.955,A -85,B 0,C 180,E1 8735.177,E2 8735.177} C_VEL
LIN {X 0,Y 586.713,Z 1097.809,A -85,B 0,C 180,E1 8739.264,E2 8739.264} C_VEL
LIN {X 0,Y 587.979,Z 1080.364,A -85,B 0,C 180,E1 8743.374,E2 8743.374} C_VEL
LIN {X 0,Y 590.083,Z 1056.999,A -85,B 0,C 180,E1 8747.512,E2 8747.512} C_VEL
LIN {X 0,Y 593.441,Z 1027.232,A -85,B 0,C 180,E1 8751.494,E2 8751.494} C_VEL
LIN {X 0,Y 597.585,Z 993.717,A -85,B 0,C 180,E1 8754.926,E2 8754.926} C_VEL
LIN {X 0,Y 601.923,Z 957.696,A -85,B 0,C 180,E1 8757.776,E2 8757.776} C_VEL
LIN {X 0,Y 606.284,Z 918.657,A -85,B 0,C 180,E1 8760.133,E2 8760.133} C_VEL
LIN {X 0,Y 610.113,Z 877.231,A -85,B 0,C 180,E1 8761.966,E2 8761.966} C_VEL
LIN {X 0,Y 612.203,Z 837.923,A -85,B 0,C 180,E1 8763.204,E2 8763.204} C_VEL
LIN {X 0,Y 593.19,Z 797.472,A -85,B 0,C 180,E1 8765.468,E2 8765.468} C_VEL
LIN {X 0,Y 585.218,Z 782.395,A -85,B 0,C 180,E1 8766.312,E2 8766.312} C_VEL
LIN {X 0,Y 585.043,Z 780.81,A -85,B 0,C 180,E1 8766.447,E2 8766.447} C_VEL
LIN {X 0,Y 585.053,Z 780.81,A -85,B 0,C 180,E1 8772.187,E2 8772.187} C_VEL
LIN {X 0,Y 585.014,Z 780.81,A -85,B 0,C 180,E1 8777.816,E2 8777.816} C_VEL
LIN {X 0,Y 585.01,Z 780.81,A -85,B 0,C 180,E1 8783.556,E2 8783.556} C_VEL
LIN {X 0,Y 585.119,Z 780.81,A -85,B 0,C 180,E1 8788.905,E2 8788.905} C_VEL
LIN {X 0,Y 585.348,Z 780.81,A -85,B 0,C 180,E1 8794.63,E2 8794.63} C_VEL
LIN {X 0,Y 585.456,Z 780.81,A -85,B 0,C 180,E1 8800.396,E2 8800.396} C_VEL
LIN {X 0,Y 585.529,Z 780.81,A -85,B 0,C 180,E1 8805.044,E2 8805.044} C_VEL
LIN {X 0,Y 585.787,Z 780.81,A -85,B 0,C 180,E1 8811.095,E2 8811.095} C_VEL
LIN {X 0,Y 586.016,Z 780.81,A -85,B 0,C 180,E1 8817.042,E2 8817.042} C_VEL
LIN {X 0,Y 586.082,Z 780.81,A -85,B 0,C 180,E1 8821.475,E2 8821.475} C_VEL
LIN {X 0,Y 585.781,Z 780.81,A -85,B 0,C 180,E1 8827.407,E2 8827.407} C_VEL
LIN {X 0,Y 585.622,Z 780.81,A -85,B 0,C 180,E1 8833.424,E2 8833.424} C_VEL
LIN {X 0,Y 585.532,Z 780.81,A -85,B 0,C 180,E1 8838.035,E2 8838.035} C_VEL
LIN {X 0,Y 585.367,Z 780.81,A -85,B 0,C 180,E1 8842.775,E2 8842.775} C_VEL
LIN {X 0,Y 585.289,Z 780.81,A -85,B 0,C 180,E1 8848.618,E2 8848.618} C_VEL
LIN {X 0,Y 585.201,Z 780.81,A -85,B 0,C 180,E1 8854.607,E2 8854.607} C_VEL
LIN {X 0,Y 584.998,Z 780.81,A -85,B 0,C 180,E1 8860.212,E2 8860.212} C_VEL
LIN {X 0,Y 584.987,Z 780.81,A -85,B 0,C 180,E1 8866.312,E2 8866.312} C_VEL
LIN {X 0,Y 585.024,Z 781.359,A -85,B 0,C 180,E1 8870.115,E2 8870.115} C_VEL
LIN {X 0,Y 613.851,Z 838.596,A -85,B 0,C 180,E1 8873.081,E2 8873.081} C_VEL
LIN {X 0,Y 612.961,Z 862.281,A -85,B 0,C 180,E1 8873.505,E2 8873.505} C_VEL
LIN {X 0,Y 608.801,Z 879.22,A -85,B 0,C 180,E1 8873.688,E2 8873.688} C_VEL
LIN {X 0,Y 604.334,Z 895.912,A -85,B 0,C 180,E1 8873.955,E2 8873.955} C_VEL
LIN {X 0,Y 600.587,Z 939.269,A -85,B 0,C 180,E1 8875.629,E2 8875.629} C_VEL
LIN {X 0,Y 596.278,Z 978.789,A -85,B 0,C 180,E1 8877.741,E2 8877.741} C_VEL
LIN {X 0,Y 591.721,Z 1016.912,A -85,B 0,C 180,E1 8880.435,E2 8880.435} C_VEL
LIN {X 0,Y 587.144,Z 1053.884,A -85,B 0,C 180,E1 8883.848,E2 8883.848} C_VEL
LIN {X 0,Y 583.34,Z 1086.208,A -85,B 0,C 180,E1 8887.737,E2 8887.737} C_VEL
LIN {X 0,Y 580.712,Z 1113.142,A -85,B 0,C 180,E1 8892,E2 8892} C_VEL
LIN {X 0,Y 579.284,Z 1132.22,A -85,B 0,C 180,E1 8896.036,E2 8896.036} C_VEL
LIN {X 0,Y 578.527,Z 1146.3,A -85,B 0,C 180,E1 8900.224,E2 8900.224} C_VEL
LIN {X 0,Y 578.29,Z 1155.689,A -85,B 0,C 180,E1 8904.752,E2 8904.752} C_VEL
LIN {X 0,Y 578.207,Z 1159.165,A -85,B 0,C 180,E1 8908.502,E2 8908.502} C_VEL
LIN {X 0,Y 578.089,Z 1158.219,A -85,B 0,C 180,E1 8912.996,E2 8912.996} C_VEL
LIN {X 0,Y 578.315,Z 1152.885,A -85,B 0,C 180,E1 8916.924,E2 8916.924} C_VEL
LIN {X 0,Y 578.705,Z 1142.004,A -85,B 0,C 180,E1 8921.23,E2 8921.23} C_VEL
LIN {X 0,Y 579.75,Z 1126.15,A -85,B 0,C 180,E1 8925.379,E2 8925.379} C_VEL
LIN {X 0,Y 581.619,Z 1104.216,A -85,B 0,C 180,E1 8929.542,E2 8929.542} C_VEL
LIN {X 0,Y 584.517,Z 1076.112,A -85,B 0,C 180,E1 8933.587,E2 8933.587} C_VEL
LIN {X 0,Y 588.731,Z 1041.312,A -85,B 0,C 180,E1 8937.412,E2 8937.412} C_VEL
LIN {X 0,Y 593.316,Z 1003.182,A -85,B 0,C 180,E1 8940.621,E2 8940.621} C_VEL
LIN {X 0,Y 598.093,Z 962.551,A -85,B 0,C 180,E1 8943.211,E2 8943.211} C_VEL
LIN {X 0,Y 602.338,Z 920.707,A -85,B 0,C 180,E1 8945.184,E2 8945.184} C_VEL
LIN {X 0,Y 605.855,Z 877.379,A -85,B 0,C 180,E1 8946.602,E2 8946.602} C_VEL
LIN {X 0,Y 607.321,Z 840.589,A -85,B 0,C 180,E1 8947.393,E2 8947.393} C_VEL
LIN {X 0,Y 585.35,Z 796.862,A -85,B 0,C 180,E1 8949.819,E2 8949.819} C_VEL
LIN {X 0,Y 577.275,Z 782.183,A -85,B 0,C 180,E1 8950.749,E2 8950.749} C_VEL
LIN {X 0,Y 577.169,Z 780.81,A -85,B 0,C 180,E1 8950.883,E2 8950.883} C_VEL
LIN {X 0,Y 577.204,Z 780.81,A -85,B 0,C 180,E1 8955.034,E2 8955.034} C_VEL
LIN {X 0,Y 577.135,Z 780.81,A -85,B 0,C 180,E1 8961.08,E2 8961.08} C_VEL
LIN {X 0,Y 577.174,Z 780.81,A -85,B 0,C 180,E1 8966.906,E2 8966.906} C_VEL
LIN {X 0,Y 577.347,Z 780.81,A -85,B 0,C 180,E1 8972.857,E2 8972.857} C_VEL
LIN {X 0,Y 577.47,Z 780.81,A -85,B 0,C 180,E1 8978.516,E2 8978.516} C_VEL
LIN {X 0,Y 577.614,Z 780.81,A -85,B 0,C 180,E1 8983.281,E2 8983.281} C_VEL
LIN {X 0,Y 577.731,Z 780.81,A -85,B 0,C 180,E1 8989.454,E2 8989.454} C_VEL
LIN {X 0,Y 577.885,Z 780.81,A -85,B 0,C 180,E1 8993.999,E2 8993.999} C_VEL
LIN {X 0,Y 578.008,Z 780.81,A -85,B 0,C 180,E1 8998.504,E2 8998.504} C_VEL
LIN {X 0,Y 577.956,Z 780.81,A -85,B 0,C 180,E1 9002.999,E2 9002.999} C_VEL
LIN {X 0,Y 577.903,Z 780.81,A -85,B 0,C 180,E1 9007.513,E2 9007.513} C_VEL
LIN {X 0,Y 577.711,Z 780.81,A -85,B 0,C 180,E1 9012.079,E2 9012.079} C_VEL
LIN {X 0,Y 577.626,Z 780.81,A -85,B 0,C 180,E1 9016.724,E2 9016.724} C_VEL
LIN {X 0,Y 577.455,Z 780.81,A -85,B 0,C 180,E1 9021.49,E2 9021.49} C_VEL
LIN {X 0,Y 577.294,Z 780.81,A -85,B 0,C 180,E1 9027.132,E2 9027.132} C_VEL
LIN {X 0,Y 577.255,Z 780.81,A -85,B 0,C 180,E1 9033.106,E2 9033.106} C_VEL
LIN {X 0,Y 577.089,Z 780.81,A -85,B 0,C 180,E1 9038.93,E2 9038.93} C_VEL
LIN {X 0,Y 577.132,Z 780.81,A -85,B 0,C 180,E1 9045.015,E2 9045.015} C_VEL
LIN {X 0,Y 577.166,Z 780.81,A -85,B 0,C 180,E1 9046.665,E2 9046.665} C_VEL
LIN {X 0,Y 579.766,Z 786.621,A -85,B 0,C 180,E1 9047.002,E2 9047.002} C_VEL
LIN {X 0,Y 600.399,Z 827.134,A -85,B 0,C 180,E1 9049.492,E2 9049.492} C_VEL
LIN {X 0,Y 606.384,Z 842.318,A -85,B 0,C 180,E1 9050.375,E2 9050.375} C_VEL
LIN {X 0,Y 603.268,Z 883.213,A -85,B 0,C 180,E1 9051.717,E2 9051.717} C_VEL
LIN {X 0,Y 599.267,Z 922.796,A -85,B 0,C 180,E1 9053.547,E2 9053.547} C_VEL
LIN {X 0,Y 594.31,Z 964.505,A -85,B 0,C 180,E1 9056.193,E2 9056.193} C_VEL
LIN {X 0,Y 589.414,Z 1002.09,A -85,B 0,C 180,E1 9059.368,E2 9059.368} C_VEL
LIN {X 0,Y 585.195,Z 1034.412,A -85,B 0,C 180,E1 9062.931,E2 9062.931} C_VEL
LIN {X 0,Y 582.16,Z 1060.744,A -85,B 0,C 180,E1 9066.682,E2 9066.682} C_VEL
LIN {X 0,Y 580.059,Z 1082.053,A -85,B 0,C 180,E1 9070.602,E2 9070.602} C_VEL
LIN {X 0,Y 578.802,Z 1099.586,A -85,B 0,C 180,E1 9074.983,E2 9074.983} C_VEL
LIN {X 0,Y 578.383,Z 1110.502,A -85,B 0,C 180,E1 9078.881,E2 9078.881} C_VEL
LIN {X 0,Y 578.046,Z 1117.668,A -85,B 0,C 180,E1 9083.339,E2 9083.339} C_VEL
LIN {X 0,Y 578.114,Z 1119.496,A -85,B 0,C 180,E1 9087.004,E2 9087.004} C_VEL
LIN {X 0,Y 578.263,Z 1116.605,A -85,B 0,C 180,E1 9091.498,E2 9091.498} C_VEL
LIN {X 0,Y 578.372,Z 1110.049,A -85,B 0,C 180,E1 9095.248,E2 9095.248} C_VEL
LIN {X 0,Y 578.881,Z 1097.958,A -85,B 0,C 180,E1 9099.391,E2 9099.391} C_VEL
LIN {X 0,Y 580.217,Z 1080.806,A -85,B 0,C 180,E1 9103.557,E2 9103.557} C_VEL
LIN {X 0,Y 582.503,Z 1057.553,A -85,B 0,C 180,E1 9107.748,E2 9107.748} C_VEL
LIN {X 0,Y 586.143,Z 1027.059,A -85,B 0,C 180,E1 9111.878,E2 9111.878} C_VEL
LIN {X 0,Y 590.74,Z 992.069,A -85,B 0,C 180,E1 9115.472,E2 9115.472} C_VEL
LIN {X 0,Y 595.652,Z 953.17,A -85,B 0,C 180,E1 9118.507,E2 9118.507} C_VEL
